# B&R Automation Studio project mappFramework (part 3)

### McBaseCfg.typ
```iecst
TYPE
	McCfgString250Type : STRING[250]; (**)
	McCfgTypeEnum :
		( (*Configuration system enum*)
		mcCFG_NONE := 0, (*None -*)
		mcCFG_MMCFG := 10, (*Associated with data type McCfgMMCfgType*)
		mcCFG_WS := 800, (*Associated with data type McCfgWorkspaceType*)
		mcCFG_TOOLTBL := 900, (*Tooltable -*)
		mcCFG_FRMTBL := 1000, (*Associated with data type McCfgFrmTblType*)
		mcCFG_DYNPARTBL := 1100, (**)
		mcCFG_TOOL := 1300, (*Tool -*)
		mcCFG_LIMSET_LIN := 1411, (*Associated with data type McCfgLimSetLinType*)
		mcCFG_LIMSET_ROT := 1412, (*Associated with data type McCfgLimSetRotType*)
		mcCFG_PROC_PT_LST := 1600, (*Associated with data type McCfgProcPtLstType*)
		mcCFG_AX := 10000, (*Associated with data type McCfgAxType*)
		mcCFG_AX_BASE_TYP := 10011, (*Associated with data type McCfgAxBaseTypType*)
		mcCFG_AX_MOVE_LIM := 10012, (*Associated with data type McCfgAxMoveLimType*)
		mcCFG_AX_FEAT_CAM_AUT_CMN := 10101, (*AxisFeatureCamAutCommon -*)
		mcCFG_AX_FEAT_PROF_GEN := 10102, (*AxisFeatureProfGen -*)
		mcCFG_AX_FEAT_DIG_CAM_SW := 10103, (*Associated with data type McCfgAxFeatDigCamSwType*)
		mcCFG_AX_FEAT_CAM_LST := 11102, (*AxisFeatureCamList -*)
		mcCFG_AX_FEAT_ALT_VAL_SRC := 10104, (*Associated with data type McCfgAxFeatAltValSrcType*)
		mcCFG_AX_FEAT_BRK := 10105, (*Associated with data type McCfgAxFeatBrkType*)
		mcCFG_AX_FEAT_MECH_DEV_COMP := 10106, (*Associated with data type McCfgAxFeatMechDevCompType*)
		mcCFG_MOT_SYN := 10500, (*Associated with data type McCfgMotSynType*)
		mcCFG_MOT_INDUCT := 10501, (*Associated with data type McCfgMotInductType*)
		mcCFG_IO_PL_IN_CARD := 10510, (*IOPlugInCard -*)
		mcCFG_ACP_AX := 11000, (*Associated with data type McCfgAcpAxType*)
		mcCFG_ACP_AX_REF := 11011, (*Associated with data type McCfgAcpAxRefType*)
		mcCFG_ACP_MECH_ELM := 11012, (*Associated with data type McCfgAcpMechElmType*)
		mcCFG_ACP_ENC_LINK := 11013, (*Associated with data type McCfgAcpEncLinkType*)
		mcCFG_ACP_CTRL := 11014, (*Associated with data type McCfgAcpCtrlType*)
		mcCFG_ACP_HOME := 11015, (*Associated with data type McCfgAcpHomeType*)
		mcCFG_ACP_STOP_REAC := 11016, (*Associated with data type McCfgAcpStopReacType*)
		mcCFG_ACP_MOVE_ERR_LIM := 11017, (*Associated with data type McCfgAcpMoveErrLimType*)
		mcCFG_ACP_JERK_FLTR := 11018, (*Associated with data type McCfgAcpJerkFltrType*)
		mcCFG_ACP_DIG_IN := 11019, (*Associated with data type McCfgAcpDigInType*)
		mcCFG_ACP_SIM := 11020, (*Associated with data type McCfgAcpSimType*)
		mcCFG_ACP_AX_FEAT := 11021, (*Associated with data type McCfgAcpAxFeatType*)
		mcCFG_ACP_AUX_PWR_SUP_MOD := 11030, (*Associated with data type McCfgAcpAuxPwrSupModType*)
		mcCFG_ACP_PSM_PWR_SEC := 11031, (*Associated with data type McCfgAcpPSMPwrSecType*)
		mcCFG_ACP_PWR_SUP := 11040, (*Associated with data type McCfgAcpPwrSupType*)
		mcCFG_ACP_ENC := 11045, (*Associated with data type McCfgAcpEncType*)
		mcCFG_ACP_VIRT_AX := 11050, (*Associated with data type McCfgAcpVirtAxType*)
		mcCFG_ACP_VIRT_AX_REF := 11051, (*Associated with data type McCfgAcpVirtAxRefType*)
		mcCFG_ACP_VIRT_HOME := 11052, (*Associated with data type McCfgAcpVirtHomeType*)
		mcCFG_ACP_VIRT_JERK_FLTR := 11053, (*Associated with data type McCfgAcpVirtJerkFltrType*)
		mcCFG_ACP_VIRT_AX_FEAT := 11054, (*Associated with data type McCfgAcpVirtAxFeatType*)
		mcCFG_ACP_CH_FEAT := 11060, (*Associated with data type McCfgAcpChFeatType*)
		mcCFG_ACP_EXT_ENC_AX := 11070, (*Associated with data type McCfgAcpExtEncAxType*)
		mcCFG_ACP_EXT_ENC_AX_REF := 11071, (*Associated with data type McCfgAcpExtEncAxRefType*)
		mcCFG_ACP_EXT_ENC_AX_ENC_LINK := 11072, (*Associated with data type McCfgAcpExtEncAxEncLinkType*)
		mcCFG_ACP_EXT_ENC_AX_MECH_ELM := 11073, (*Associated with data type McCfgAcpExtEncAxMechElmType*)
		mcCFG_ACP_EXT_ENC_AX_HOME := 11074, (*Associated with data type McCfgAcpExtEncAxHomeType*)
		mcCFG_AX_FEAT_CAM_AUT_ACP := 11101, (*AxisFeatureCamAutAcopos -*)
		mcCFG_AX_FEAT_A_IN := 11103, (*AxisFeatureAInput -*)
		mcCFG_AX_FEAT_ACP_PAR_TBL := 11104, (*Associated with data type McCfgAxFeatAcpParTblType*)
		mcCFG_PURE_V_AX := 12000, (*Associated with data type McCfgPureVAxType*)
		mcCFG_PURE_V_AX_REF := 12011, (*Associated with data type McCfgPureVAxRefType*)
		mcCFG_PURE_V_AX_HOME := 12012, (*Associated with data type McCfgPureVAxHomeType*)
		mcCFG_PURE_V_AX_JERK_FLTR := 12013, (*Associated with data type McCfgPureVAxJerkFltrType*)
		mcCFG_PURE_V_AX_FEAT := 12014, (*Associated with data type McCfgPureVAxFeatType*)
		mcCFG_PURE_V_AX_MECH_ELM := 12015, (*Associated with data type McCfgPureVAxMechElmType*)
		mcCFG_PURE_V_AX_ENC_LINK := 12016, (*Associated with data type McCfgPureVAxEncLinkType*)
		mcCFG_PURE_V_AX_CTRL := 12017, (*Associated with data type McCfgPureVAxCtrlType*)
		mcCFG_PURE_V_AX_STOP_REAC := 12018, (*Associated with data type McCfgPureVAxStopReacType*)
		mcCFG_PURE_V_AX_MOVE_ERR_LIM := 12019, (*Associated with data type McCfgPureVAxMoveErrLimType*)
		mcCFG_PURE_V_AX_DIG_IN := 12020, (*Associated with data type McCfgPureVAxDigInType*)
		mcCFG_PURE_V_AX_STAT_IN := 12021, (*Associated with data type McCfgPureVAxStatInType*)
		mcCFG_PURE_V_AX_CTRL_OUT := 12022, (*Associated with data type McCfgPureVAxCtrlOutType*)
		mcCFG_STP_AX := 13000, (*Associated with data type McCfgStpAxType*)
		mcCFG_STP_AX_REF := 13011, (*Associated with data type McCfgStpAxRefType*)
		mcCFG_STP_AX_MECH_ELM := 13012, (*Associated with data type McCfgStpAxMechElmType*)
		mcCFG_STP_AX_MOT := 13013, (*Associated with data type McCfgStpAxMotType*)
		mcCFG_STP_AX_ENC_LINK := 13014, (*Associated with data type McCfgStpAxEncLinkType*)
		mcCFG_STP_AX_CTRL := 13015, (*Associated with data type McCfgStpAxCtrlType*)
		mcCFG_STP_AX_HOME := 13016, (*Associated with data type McCfgStpAxHomeType*)
		mcCFG_STP_AX_STOP_REAC := 13017, (*Associated with data type McCfgStpAxStopReacType*)
		mcCFG_STP_AX_MOVE_ERR_LIM := 13018, (*Associated with data type McCfgStpAxMoveErrLimType*)
		mcCFG_STP_AX_JERK_FLTR := 13019, (*Associated with data type McCfgStpAxJerkFltrType*)
		mcCFG_STP_AX_DIG_IN := 13020, (*Associated with data type McCfgStpAxDigInType*)
		mcCFG_STP_AX_DIG_OUT := 13021, (*Associated with data type McCfgStpAxDigOutType*)
		mcCFG_STP_AX_FEAT := 13022, (*Associated with data type McCfgStpAxFeatType*)
		mcCFG_STP_ENC := 13100, (*Associated with data type McCfgStpEncType*)
		mcCFG_DS402_AX := 13500, (*Associated with data type McCfgDS402AxType*)
		mcCFG_DS402_INV_AX := 13501, (*Associated with data type McCfgDS402InvAxType*)
		mcCFG_DS402_AX_REF := 13511, (*Associated with data type McCfgDS402AxRefType*)
		mcCFG_DS402_AX_MECH_ELM := 13512, (*Associated with data type McCfgDS402AxMechElmType*)
		mcCFG_DS402_AX_ENC_SET := 13513, (*Associated with data type McCfgDS402AxEncSetType*)
		mcCFG_DS402_AX_POS_ACT_VAL_RNG := 13514, (*Associated with data type McCfgDS402AxPosActValRngType*)
		mcCFG_DS402_AX_CYC_SET_VAL_MOD := 13515, (*Associated with data type McCfgDS402AxCycSetValModType*)
		mcCFG_DS402_AX_FEAT := 13516, (*Associated with data type McCfgDS402AxFeatType*)
		mcCFG_ACP_INV_AX := 13600, (*Associated with data type McCfgAcpInvAxType*)
		mcCFG_ACP_INV_AX_REF := 13611, (*Associated with data type McCfgAcpInvAxRefType*)
		mcCFG_ACP_INV_AX_MECH_ELM := 13612, (*Associated with data type McCfgAcpInvAxMechElmType*)
		mcCFG_AXGRP_ADMIN := 20000, (*Associated with data type McCfgAxGrpAdminType*)
		mcCFG_AXGRP_FEAT_HOME_ORD := 20101, (*Associated with data type McCfgAxGrpFeatHomeOrdType*)
		mcCFG_AXGRP_FEAT_PWR_ON_ORD := 20102, (*Associated with data type McCfgAxGrpFeatPwrOnOrdType*)
		mcCFG_AXGRP_FEAT_EX_SNG_AX := 20103, (*Associated with data type McCfgAxGrpFeatExSngAxType*)
		mcCFG_AXGRP_FEAT_SHR_BRK_SIG := 20104, (*Associated with data type McCfgAxGrpFeatShrBrkSigType*)
		mcCFG_AXGRP_PATHGEN := 21000, (*Associated with data type McCfgAxGrpPathGenType*)
		mcCFG_AXGRP_PATHGEN_BASE_SET := 21013, (*Associated with data type McCfgAxGrpPathGenBaseSetType*)
		mcCFG_AXGRP_FEAT_PRG := 21101, (*Associated with data type McCfgAxGrpFeatPrgType*)
		mcCFG_AXGRP_FEAT_COMP := 21102, (*Associated with data type McCfgAxGrpFeatCompType*)
		mcCFG_AXGRP_FEAT_CDC := 21103, (*Associated with data type McCfgAxGrpFeatCdcType*)
		mcCFG_AXGRP_FEAT_FF := 21104, (*Associated with data type McCfgAxGrpFeatFfType*)
		mcCFG_AXGRP_FEAT_FRM_HIER_STD := 21105, (*Associated with data type McCfgAxGrpFeatFrmHierStdType*)
		mcCFG_AXGRP_FEAT_FRM_HIER_CUS := 21106, (*Associated with data type McCfgAxGrpFeatFrmHierCusType*)
		mcCFG_AXGRP_FEAT_JOG := 21107, (*AxesgroupFeatureJogging -*)
		mcCFG_AXGRP_FEAT_LAH := 21108, (*Associated with data type McCfgAxGrpFeatLahType*)
		mcCFG_AXGRP_FEAT_MFUN := 21109, (*Associated with data type McCfgAxGrpFeatMFunType*)
		mcCFG_AXGRP_FEAT_MON_ELEM := 21110, (*Associated with data type McCfgAxGrpFeatMonElemType*)
		mcCFG_AXGRP_FEAT_MP_LOG := 21111, (*Associated with data type McCfgAxGrpFeatMpLogType*)
		mcCFG_AXGRP_FEAT_PATH_DEF := 21112, (*Associated with data type McCfgAxGrpFeatPathDefType*)
		mcCFG_AXGRP_FEAT_PRG_SIM := 21113, (*Associated with data type McCfgAxGrpFeatPrgSimType*)
		mcCFG_AXGRP_FEAT_SPINDLES := 21114, (*Associated with data type McCfgAxGrpFeatSpindlesType*)
		mcCFG_AXGRP_FEAT_TOOL := 21115, (*Associated with data type McCfgAxGrpFeatToolType*)
		mcCFG_AXGRP_FEAT_WSM := 21116, (*Associated with data type McCfgAxGrpFeatWsmType*)
		mcCFG_AXGRP_FEAT_EX_PATH_AX := 21117, (*Associated with data type McCfgAxGrpFeatExPathAxType*)
		mcCFG_AXGRP_FEAT_PROBE := 21118, (*Associated with data type McCfgAxGrpFeatProbeType*)
		mcCFG_AXGRP_FEAT_SIG := 21119, (*Associated with data type McCfgAxGrpFeatSigType*)
		mcCFG_AXGRP_FEAT_2D_COMP := 21120, (*Associated with data type McCfgAxGrpFeat2DCompType*)
		mcCFG_AXGRP_FEAT_3D_COMP := 21121, (*Associated with data type McCfgAxGrpFeat3DCompType*)
		mcCFG_AXGRP_FEAT_PATH_PREVIEW := 21122, (*Associated with data type McCfgAxGrpFeatPathPreviewType*)
		mcCFG_AXGRP_FEAT_TAN_TOOL := 21124, (*Associated with data type McCfgAxGrpFeatTanToolType*)
		mcCFG_AXGRP_FEAT_REV_MOVE := 21125, (*Associated with data type McCfgAxGrpFeatRevMoveType*)
		mcCFG_ASM := 31000, (*Associated with data type McCfgAsmType*)
		mcCFG_ASM_FEAT_CPLG := 31101, (*Associated with data type McCfgAsmFeatCplgType*)
		mcCFG_ASM_FEAT_SIM_SH_DEF := 31102, (*Associated with data type McCfgAsmFeatSimShDefType*)
		mcCFG_ASM_FEAT_SH_TRACE := 31103, (*Associated with data type McCfgAsmFeatShTraceType*)
		mcCFG_ASM_FEAT_SH_AUT_ATT := 31104, (*Associated with data type McCfgAsmFeatShAutAttType*)
		mcCFG_ASM_FEAT_LOC_LIM := 31105, (*Associated with data type McCfgAsmFeatLocLimType*)
		mcCFG_ASM_FEAT_EX_SEG := 31106, (*Associated with data type McCfgAsmFeatExSegType*)
		mcCFG_ASM_FEAT_SH_SHP_REG := 31107, (*Associated with data type McCfgAsmFeatShShpRegType*)
		mcCFG_SEC_COMP := 31301, (*Associated with data type McCfgSecCompType*)
		mcCFG_SEC_SUB := 31302, (*Associated with data type McCfgSecSubType*)
		mcCFG_SH_STEREO_TYP := 31400, (*Associated with data type McCfgShStereoTypType*)
		mcCFG_SEG := 31500, (*Associated with data type McCfgSegType*)
		mcCFG_MS_CUS_STD := 50001, (*Associated with data type McCfgMSCusStdType*)
		mcCFG_MS_2AX_CNC_XY := 51201, (*Associated with data type McCfgMS2AxCncXYType*)
		mcCFG_MS_2AX_CNC_XZ := 51202, (*Associated with data type McCfgMS2AxCncXZType*)
		mcCFG_MS_2AX_CNC_YZ := 51203, (*Associated with data type McCfgMS2AxCncYZType*)
		mcCFG_MS_3AX_CNC_XYZ := 51301, (*Associated with data type McCfgMS3AxCncXYZType*)
		mcCFG_MS_3AX_CNC_XZC := 51302, (*Associated with data type McCfgMS3AxCncXZCType*)
		mcCFG_MS_3AX_CNC_XZB := 51303, (*Associated with data type McCfgMS3AxCncXZBType*)
		mcCFG_MS_4AX_CNC_XYZB := 51401, (*Associated with data type McCfgMS4AxCncXYZBType*)
		mcCFG_MS_4AX_CNC_XYZC := 51402, (*Associated with data type McCfgMS4AxCncXYZCType*)
		mcCFG_MS_5AX_CNC_XYZCA := 51504, (*Associated with data type McCfgMS5AxCncXYZCAType*)
		mcCFG_MS_6AX_CNC_ZXYBCA := 51603, (*Associated with data type McCfgMS6AxCncZXYBCAType*)
		mcCFG_MS_4AX_SCARA_A := 52041, (*Associated with data type McCfgMS4AxScaraAType*)
		mcCFG_MS_2AX_DELTA_A := 52121, (*Associated with data type McCfgMS2AxDeltaAType*)
		mcCFG_MS_3AX_DELTA_A := 52131, (*Associated with data type McCfgMS3AxDeltaAType*)
		mcCFG_MS_3AX_DELTA_XZB := 52132, (*Associated with data type McCfgMS3AxDeltaXZBType*)
		mcCFG_MS_3AX_DELTA_B := 52133, (*Associated with data type McCfgMS3AxDeltaBType*)
		mcCFG_MS_4AX_DELTA_A := 52141, (*Associated with data type McCfgMS4AxDeltaAType*)
		mcCFG_MS_4AX_DELTA_B := 52142, (*Associated with data type McCfgMS4AxDeltaBType*)
		mcCFG_MS_4AX_DELTA_C := 52143, (*Associated with data type McCfgMS4AxDeltaCType*)
		mcCFG_MS_5AX_DELTA_A := 52151, (*Associated with data type McCfgMS5AxDeltaAType*)
		mcCFG_MS_3AX_ROB_A := 52301, (*Associated with data type McCfgMS3AxRobAType*)
		mcCFG_MS_4AX_ROB_A := 52401, (*Associated with data type McCfgMS4AxRobAType*)
		mcCFG_MS_4AX_ROB_B := 52402, (*Associated with data type McCfgMS4AxRobBType*)
		mcCFG_MS_5AX_ROB_A := 52501, (*Associated with data type McCfgMS5AxRobAType*)
		mcCFG_MS_5AX_ROB_B := 52502, (*Associated with data type McCfgMS5AxRobBType*)
		mcCFG_MS_6AX_ROB_A := 52601, (*Associated with data type McCfgMS6AxRobAType*)
		mcCFG_MS_6AX_ROB_B := 52602, (*Associated with data type McCfgMS6AxRobBType*)
		mcCFG_MS_6AX_ROB_C := 52603 (*Associated with data type McCfgMS6AxRobCType*)
		);
	McCfgUnboundedArrayType : STRUCT (*General purpose datatype*)
		NumberOfElements : UDINT;
		DataAddress : UDINT;
		NumberOfArrayElements : UDINT;
	END_STRUCT;
	McCfgReferenceType : STRUCT (*General purpose datatype*)
		Name : STRING[250];
		ConfigType : McCfgTypeEnum;
	END_STRUCT;
	McMMCProcProcTskCEnum :
		( (*Cyclic task class for command processing*)
		mcMMCPPTC_CYC_1 := 1, (*Cyclic #1 - Task class 1*)
		mcMMCPPTC_CYC_2 := 2 (*Cyclic #2 - Task class 2*)
		);
	McMMCProcType : STRUCT
		ProcessingTaskClass : McMMCProcProcTskCEnum; (*Cyclic task class for command processing*)
	END_STRUCT;
	McMMCLogSelEnum :
		( (*Selective logging selector setting*)
		mcMMCLS_NOT_USE := 0, (*Not used -*)
		mcMMCLS_USE := 1 (*Used -*)
		);
	McCfgVisEnum :
		( (*Component state change logger entries (PLCopen state)*)
		mcCV_VIS := 0, (*Visible*)
		mcCV_SUP := 1 (*Suppressed*)
		);
	McMMCLogSelUseAdmCmdEnum :
		( (*Administrative commands selector setting*)
		mcMMCLSUAC_VIS := 0, (*Visible - This command group of logger entries will be visible*)
		mcMMCLSUAC_SUP := 1, (*Suppressed - This command group of logger entries will be suppressed*)
		mcMMCLSUAC_SEL := 2 (*Selective - Defines which sections of this command group should be visible*)
		);
	McMMCLogSelUseAdmCmdSelType : STRUCT (*Type mcMMCLSUAC_SEL settings*)
		CallerInstance : McCfgVisEnum; (*Logging of the caller instance entries*)
		ComponentResponse : McCfgVisEnum; (*Logging of component response entries*)
		AdditionalInformation : McCfgVisEnum; (*Logging of additional information entries*)
	END_STRUCT;
	McMMCLogSelUseAdmCmdType : STRUCT (*Administrative logger entries*)
		Type : McMMCLogSelUseAdmCmdEnum; (*Administrative commands selector setting*)
		Selective : McMMCLogSelUseAdmCmdSelType; (*Type mcMMCLSUAC_SEL settings*)
	END_STRUCT;
	McMMCLogSelUseMoveCmdEnum :
		( (*Movement commands selector setting*)
		mcMMCLSUMC_VIS := 0, (*Visible - This command group of logger entries will be visible*)
		mcMMCLSUMC_SUP := 1, (*Suppressed - This command group of logger entries will be suppressed*)
		mcMMCLSUMC_SEL := 2 (*Selective - Defines which sections of this command group should be visible*)
		);
	McMMCLogSelUseMoveCmdSelType : STRUCT (*Type mcMMCLSUMC_SEL settings*)
		CallerInstance : McCfgVisEnum; (*Logging of the caller instance entries*)
		ComponentResponse : McCfgVisEnum; (*Logging of component response entries*)
		AdditionalInformation : McCfgVisEnum; (*Logging of additional information entries*)
	END_STRUCT;
	McMMCLogSelUseMoveCmdType : STRUCT (*Movement logger entries*)
		Type : McMMCLogSelUseMoveCmdEnum; (*Movement commands selector setting*)
		Selective : McMMCLogSelUseMoveCmdSelType; (*Type mcMMCLSUMC_SEL settings*)
	END_STRUCT;
	McMMCLogSelUseInfoCmdEnum :
		( (*Informational commands selector setting*)
		mcMMCLSUIC_VIS := 0, (*Visible - This command group of logger entries will be visible*)
		mcMMCLSUIC_SUP := 1, (*Suppressed - This command group of logger entries will be suppressed*)
		mcMMCLSUIC_SEL := 2 (*Selective - Defines which sections of this command group should be visible*)
		);
	McMMCLogSelUseInfoCmdSelType : STRUCT (*Type mcMMCLSUIC_SEL settings*)
		CallerInstance : McCfgVisEnum; (*Logging of the caller instance entries*)
		ComponentResponse : McCfgVisEnum; (*Logging of component response entries*)
		AdditionalInformation : McCfgVisEnum; (*Logging of additional information entries*)
	END_STRUCT;
	McMMCLogSelUseInfoCmdType : STRUCT (*Status information logger entries*)
		Type : McMMCLogSelUseInfoCmdEnum; (*Informational commands selector setting*)
		Selective : McMMCLogSelUseInfoCmdSelType; (*Type mcMMCLSUIC_SEL settings*)
	END_STRUCT;
	McMMCLogSelUseSupSubcEEnum :
		( (*Suppress entries for internally invoked commands for subcomponents*)
		mcMMCLSUSSE_INACT := 0, (*Inactive - Entries for internally invoked commands for subcomponents are shown unless the base entries are suppressed*)
		mcMMCLSUSSE_ACT := 1 (*Active - Entries for internally invoked commands for subcomponents are suppressed*)
		);
	McMMCLogSelUseType : STRUCT (*Type mcMMCLS_USE settings*)
		StateChange : McCfgVisEnum; (*Component state change logger entries (PLCopen state)*)
		AdministrativeCommands : McMMCLogSelUseAdmCmdType; (*Administrative logger entries*)
		MovementCommands : McMMCLogSelUseMoveCmdType; (*Movement logger entries*)
		InformationalCommands : McMMCLogSelUseInfoCmdType; (*Status information logger entries*)
		SuppressSubcomponentEntries : McMMCLogSelUseSupSubcEEnum; (*Suppress entries for internally invoked commands for subcomponents*)
	END_STRUCT;
	McMMCLogSelType : STRUCT (*Define which logging areas should be visible*)
		Type : McMMCLogSelEnum; (*Selective logging selector setting*)
		Used : McMMCLogSelUseType; (*Type mcMMCLS_USE settings*)
	END_STRUCT;
	McMMCLogType : STRUCT
		Selective : McMMCLogSelType; (*Define which logging areas should be visible*)
	END_STRUCT;
	McCfgMMCfgType : STRUCT (*Main data type corresponding to McCfgTypeEnum mcCFG_MMCFG*)
		Processing : McMMCProcType;
		Logger : McMMCLogType;
	END_STRUCT;
	McCfgTransXYZType : STRUCT (*Translation parameters*)
		X : LREAL; (*Translation in X direction [measurement units]*)
		Y : LREAL; (*Translation in Y direction [measurement units]*)
		Z : LREAL; (*Translation in Z direction [measurement units]*)
	END_STRUCT;
	McCfgOrientType : STRUCT (*Orientation parameters*)
		Angle1 : LREAL; (*Rotation around the first coordinateaxis of the rotation order [measurement units]*)
		Angle2 : LREAL; (*Rotation around the second coordinateaxis of the rotation order [measurement units]*)
		Angle3 : LREAL; (*Rotation around the third coordinateaxis of the rotation order [measurement units]*)
	END_STRUCT;
	McWSCubeDimType : STRUCT (*Dimension parameters*)
		X : LREAL; (*Dimension of the cuboid in the x-direction (endpoint) [measurement units]*)
		Y : LREAL; (*Dimension of the cuboid in the y-direction (endpoint) [measurement units]*)
		Z : LREAL; (*Dimension of the cuboid in the z-direction (endpoint) [measurement units]*)
	END_STRUCT;
	McWSCubeType : STRUCT
		ID : UDINT; (*Unique cuboid ID*)
		Translation : McCfgTransXYZType; (*Translation parameters*)
		Orientation : McCfgOrientType; (*Orientation parameters*)
		Dimension : McWSCubeDimType; (*Dimension parameters*)
	END_STRUCT;
	McWSCubesType : STRUCT (*Defines cuboids*)
		Cuboid : McCfgUnboundedArrayType;
	END_STRUCT;
	McWSHalfSpcPlEnum :
		( (*Defines plane*)
		mcWSHSP_PL_XY := 0, (*Plane XY*)
		mcWSHSP_PL_YZ := 1, (*Plane YZ*)
		mcWSHSP_PL_ZX := 2 (*Plane ZX*)
		);
	McWSHalfSpcType : STRUCT
		ID : UDINT; (*Unique half-space ID*)
		Translation : McCfgTransXYZType; (*Translation parameters*)
		Orientation : McCfgOrientType; (*Orientation parameters*)
		Plane : McWSHalfSpcPlEnum; (*Defines plane*)
	END_STRUCT;
	McWSHalfSpcsType : STRUCT (*Defines half-spaces*)
		HalfSpace : McCfgUnboundedArrayType;
	END_STRUCT;
	McWSTcConeParType : STRUCT (*Object description parameters*)
		BaseRadius : LREAL; (*Base radius of the cone [measurement units]*)
		Height : LREAL; (*Height of the cone [measurement units]*)
		TopRadius : LREAL; (*Top radius of the cone [measurement units]*)
	END_STRUCT;
	McWSTcConeType : STRUCT (*Selects object type*)
		ID : UDINT; (*Unique object ID*)
		Translation : McCfgTransXYZType; (*Translation parameters*)
		Orientation : McCfgOrientType; (*Orientation parameters*)
		Parameters : McWSTcConeParType; (*Object description parameters*)
	END_STRUCT;
	McWSTcConesType : STRUCT (*Defines truncated cones*)
		TruncatedCone : McCfgUnboundedArrayType; (*Selects object type*)
	END_STRUCT;
	McWSWorkSpaceType : STRUCT (*Defines the WorkSpace*)
		Cuboids : McWSCubesType; (*Defines cuboids*)
		HalfSpaces : McWSHalfSpcsType; (*Defines half-spaces*)
		TruncatedCones : McWSTcConesType; (*Defines truncated cones*)
	END_STRUCT;
	McWSSafeSpaceType : STRUCT (*Defines the SafeSpace*)
		Cuboids : McWSCubesType; (*Defines cuboids*)
		HalfSpaces : McWSHalfSpcsType; (*Defines half-spaces*)
		TruncatedCones : McWSTcConesType; (*Defines truncated cones*)
	END_STRUCT;
	McCfgWorkspaceType : STRUCT (*Main data type corresponding to McCfgTypeEnum mcCFG_WS*)
		WorkSpace : McWSWorkSpaceType; (*Defines the WorkSpace*)
		SafeSpace : McWSSafeSpaceType; (*Defines the SafeSpace*)
	END_STRUCT;
	McFTRowType : STRUCT
		Index : UINT;
		X : LREAL;
		Y : LREAL;
		Z : LREAL;
		Angle1 : LREAL;
		Angle2 : LREAL;
		Angle3 : LREAL;
		Description : STRING[250];
	END_STRUCT;
	McCfgFrmTblType : STRUCT (*Main data type corresponding to McCfgTypeEnum mcCFG_FRMTBL*)
		Row : McCfgUnboundedArrayType;
	END_STRUCT;
	McLSPosEnum :
		( (*Position selector setting*)
		mcLSP_NOT_USE := 0, (*Not used -*)
		mcLSP_USE := 1 (*Used -*)
		);
	McCfgLimPosType : STRUCT (*Type mcLSP_USE settings*)
		LowerLimit : LREAL; (*Lower software limit position [Measurement units]*)
		UpperLimit : LREAL; (*Upper software limit position [Measurement units]*)
	END_STRUCT;
	McLSPosType : STRUCT (*Movement range of the axis via two position boundaries*)
		Type : McLSPosEnum; (*Position selector setting*)
		Used : McCfgLimPosType; (*Type mcLSP_USE settings*)
	END_STRUCT;
	McLSVelEnum :
		( (*Velocity selector setting*)
		mcLSV_NOT_USE := 0, (*Not used -*)
		mcLSV_BASIC := 1, (*Basic -*)
		mcLSV_ADV := 2 (*Advanced -*)
		);
	McCfgLimVelBaseType : STRUCT (*Type mcLSV_BASIC settings*)
		Velocity : REAL; (*Velocity limit in any movement direction [Measurement units/s]*)
	END_STRUCT;
	McCfgLimVelAdvType : STRUCT (*Type mcLSV_ADV settings*)
		Positive : REAL; (*Velocity limit in positive movement direction [Measurement units/s]*)
		Negative : REAL; (*Velocity limit in negative movement direction [Measurement units/s]*)
	END_STRUCT;
	McLSVelType : STRUCT (*Velocity limits*)
		Type : McLSVelEnum; (*Velocity selector setting*)
		Basic : McCfgLimVelBaseType; (*Type mcLSV_BASIC settings*)
		Advanced : McCfgLimVelAdvType; (*Type mcLSV_ADV settings*)
	END_STRUCT;
	McLSAccEnum :
		( (*Acceleration selector setting*)
		mcLSA_NOT_USE := 0, (*Not used -*)
		mcLSA_BASIC := 1, (*Basic -*)
		mcLSA_ADV := 2 (*Advanced -*)
		);
	McCfgLimAccBaseType : STRUCT (*Type mcLSA_BASIC settings*)
		Acceleration : REAL; (*Acceleration limit in any movement direction [Measurement units/s²]*)
	END_STRUCT;
	McCfgLimAccAdvType : STRUCT (*Type mcLSA_ADV settings*)
		Positive : REAL; (*Acceleration limit in positive movement direction [Measurement units/s²]*)
		Negative : REAL; (*Acceleration limit in negative movement direction [Measurement units/s²]*)
	END_STRUCT;
	McLSAccType : STRUCT (*Acceleration limits*)
		Type : McLSAccEnum; (*Acceleration selector setting*)
		Basic : McCfgLimAccBaseType; (*Type mcLSA_BASIC settings*)
		Advanced : McCfgLimAccAdvType; (*Type mcLSA_ADV settings*)
	END_STRUCT;
	McLSDecEnum :
		( (*Deceleration selector setting*)
		mcLSD_NOT_USE := 0, (*Not used -*)
		mcLSD_BASIC := 1, (*Basic -*)
		mcLSD_ADV := 2 (*Advanced -*)
		);
	McCfgLimDecBaseType : STRUCT (*Type mcLSD_BASIC settings*)
		Deceleration : REAL; (*Deceleration limit in any movement direction [Measurement units/s²]*)
	END_STRUCT;
	McCfgLimDecAdvType : STRUCT (*Type mcLSD_ADV settings*)
		Positive : REAL; (*Deceleration limit in positive movement direction [Measurement units/s²]*)
		Negative : REAL; (*Deceleration limit in negative movement direction [Measurement units/s²]*)
	END_STRUCT;
	McLSDecType : STRUCT (*Deceleration limits*)
		Type : McLSDecEnum; (*Deceleration selector setting*)
		Basic : McCfgLimDecBaseType; (*Type mcLSD_BASIC settings*)
		Advanced : McCfgLimDecAdvType; (*Type mcLSD_ADV settings*)
	END_STRUCT;
	McCfgLimJerkEnum :
		( (*Jerk selector setting*)
		mcCLJ_NOT_USE := 0, (*Not used -*)
		mcCLJ_BASIC := 1, (*Basic -*)
		mcCLJ_ADV := 2 (*Advanced -*)
		);
	McCfgLimJerkBasicType : STRUCT (*Type mcCLJ_BASIC settings*)
		Jerk : REAL; (*Jerk limit in any movement direction [Measurement units/s³]*)
	END_STRUCT;
	McCfgLimJerkAdvType : STRUCT (*Type mcCLJ_ADV settings*)
		AccelerationPositive : REAL; (*Jerk limit in positive movement direction during acceleration [Measurement units/s³]*)
		AccelerationNegative : REAL; (*Jerk limit in negative movement direction during acceleration [Measurement units/s³]*)
		DecelerationPositive : REAL; (*Jerk limit in positive movement direction during deceleration [Measurement units/s³]*)
		DecelerationNegative : REAL; (*Jerk limit in negative movement direction during deceleration [Measurement units/s³]*)
	END_STRUCT;
	McCfgLimJerkType : STRUCT (*Jerk limits*)
		Type : McCfgLimJerkEnum; (*Jerk selector setting*)
		Basic : McCfgLimJerkBasicType; (*Type mcCLJ_BASIC settings*)
		Advanced : McCfgLimJerkAdvType; (*Type mcCLJ_ADV settings*)
	END_STRUCT;
	McCfgLimForEnum :
		( (*Force selector setting*)
		mcCLF_NOT_USE := 0, (*Not used -*)
		mcCLF_BASIC := 1, (*Basic -*)
		mcCLF_ADV := 2 (*Advanced -*)
		);
	McCfgLimForBasicType : STRUCT (*Type mcCLF_BASIC settings*)
		Force : REAL; (*Force limit in any movement direction [N]*)
	END_STRUCT;
	McCfgLimForAdvType : STRUCT (*Type mcCLF_ADV settings*)
		AccelerationPositive : REAL; (*Force limit in positive movement direction during acceleration [N]*)
		AccelerationNegative : REAL; (*Force limit in negative movement direction during acceleration [N]*)
		DecelerationPositive : REAL; (*Force limit in positive movement direction during deceleration [N]*)
		DecelerationNegative : REAL; (*Force limit in negative movement direction during deceleration [N]*)
	END_STRUCT;
	McCfgLimForType : STRUCT (*Limits for the force of the axis*)
		Type : McCfgLimForEnum; (*Force selector setting*)
		Basic : McCfgLimForBasicType; (*Type mcCLF_BASIC settings*)
		Advanced : McCfgLimForAdvType; (*Type mcCLF_ADV settings*)
	END_STRUCT;
	McCfgLimSetLinType : STRUCT (*Main data type corresponding to McCfgTypeEnum mcCFG_LIMSET_LIN*)
		Position : McLSPosType; (*Movement range of the axis via two position boundaries*)
		Velocity : McLSVelType; (*Velocity limits*)
		Acceleration : McLSAccType; (*Acceleration limits*)
		Deceleration : McLSDecType; (*Deceleration limits*)
		Jerk : McCfgLimJerkType; (*Jerk limits*)
		Force : McCfgLimForType; (*Limits for the force of the axis*)
	END_STRUCT;
	McCfgLimTorqEnum :
		( (*Torque selector setting*)
		mcCLT_NOT_USE := 0, (*Not used -*)
		mcCLT_BASIC := 1, (*Basic -*)
		mcCLT_ADV := 2 (*Advanced -*)
		);
	McCfgLimTorqBasicType : STRUCT (*Type mcCLT_BASIC settings*)
		Torque : REAL; (*Torque limit in any movement direction [Nm]*)
	END_STRUCT;
	McCfgLimTorqAdvType : STRUCT (*Type mcCLT_ADV settings*)
		AccelerationPositive : REAL; (*Torque limit in positive movement direction during acceleration [Nm]*)
		AccelerationNegative : REAL; (*Torque limit in negative movement direction during acceleration [Nm]*)
		DecelerationPositive : REAL; (*Torque limit in positive movement direction during deceleration [Nm]*)
		DecelerationNegative : REAL; (*Torque limit in negative movement direction during deceleration [Nm]*)
	END_STRUCT;
	McCfgLimTorqType : STRUCT (*Torque limits*)
		Type : McCfgLimTorqEnum; (*Torque selector setting*)
		Basic : McCfgLimTorqBasicType; (*Type mcCLT_BASIC settings*)
		Advanced : McCfgLimTorqAdvType; (*Type mcCLT_ADV settings*)
	END_STRUCT;
	McCfgLimSetRotType : STRUCT (*Main data type corresponding to McCfgTypeEnum mcCFG_LIMSET_ROT*)
		Position : McLSPosType; (*Movement range of the axis via two position boundaries*)
		Velocity : McLSVelType; (*Velocity limits*)
		Acceleration : McLSAccType; (*Acceleration limits*)
		Deceleration : McLSDecType; (*Deceleration limits*)
		Jerk : McCfgLimJerkType; (*Jerk limits*)
		Torque : McCfgLimTorqType; (*Torque limits*)
	END_STRUCT;
	McPPLPtEnum :
		( (*Process point: {/} selector setting*)
		mcPPLP_TRAK_PT := 0 (*Trak point - ACOPOSTrak*)
		);
	McPPLPtTrakPtPosRelToEnum :
		( (*Absolute position from which the position is counted*)
		mcPPLPTPPRT_ST_OF_SEC := 0, (*Start of sector - Tail of the sector*)
		mcPPLPTPPRT_END_OF_SEC := 1 (*End of sector - Head of the sector*)
		);
	McPPLPtTrakPtBarrFunEnum :
		( (*Barrier functionality selector setting*)
		mcPPLPTPBF_OFF := 0, (*Off - Disable barrier functionality*)
		mcPPLPTPBF_ON := 1 (*On - Enable barrier functionality*)
		);
	McPPLPtTrakPtBarrFunType : STRUCT (*Enable barrier functionality for process point*)
		Type : McPPLPtTrakPtBarrFunEnum; (*Barrier functionality selector setting*)
	END_STRUCT;
	McPPLPtTrakPtType : STRUCT (*Type mcPPLP_TRAK_PT settings*)
		Name : STRING[250]; (*Identifier of point*)
		SectorReference : McCfgReferenceType; (*Name of the referenced sector component*)
		Position : LREAL; (*Position on the sector [Measurement units]*)
		PositionRelativeTo : McPPLPtTrakPtPosRelToEnum; (*Absolute position from which the position is counted*)
		TriggerEventBufferSize : UINT; (*Amount of maximum saved trigger point events*)
		BarrierFunctionality : McPPLPtTrakPtBarrFunType; (*Enable barrier functionality for process point*)
	END_STRUCT;
	McPPLPtType : STRUCT
		Type : McPPLPtEnum; (*Process point: {/} selector setting*)
		TrakPoint : McPPLPtTrakPtType; (*Type mcPPLP_TRAK_PT settings*)
	END_STRUCT;
	McCfgProcPtLstType : STRUCT (*Main data type corresponding to McCfgTypeEnum mcCFG_PROC_PT_LST*)
		ProcessPoints : McCfgUnboundedArrayType;
	END_STRUCT;
	McCfgLocLenUnitEnum :
		( (*Measurement unit for the axis*)
		mcCLLU_G_SET := 0, (*Global settings*)
		mcCLLU_MILL := 5066068, (*Millimeters*)
		mcCLLU_M := 5067858, (*Meters*)
		mcCLLU_INCH := 4804168, (*Inches*)
		mcCLLU_GEN := -1 (*Generic*)
		);
	McCfgCntDirEnum :
		( (*Direction of the axis in which the position value is increasing*)
		mcCCD_STD := 0, (*Standard - Rotary axis: clockwise*)
		mcCCD_INV := 1 (*Inverse - Rotary axis: counter-clockwise*)
		);
	McCfgLocRotUnitEnum :
		( (*Measurement unit for the axis*)
		mcCLRU_G_SET := 0, (*Global settings*)
		mcCLRU_DEG := 17476, (*Degrees*)
		mcCLRU_GRAD := 4274481, (*Gradians*)
		mcCLRU_REV := 5059636, (*Revolutions*)
		mcCLRU_GEN := -1 (*Generic*)
		);
	McCfgExtLimRefType : STRUCT (*Type mcAML_EXT settings*)
		LimitReference : McCfgReferenceType; (*Name of the limit reference*)
	END_STRUCT;
	McCfgGearBoxType : STRUCT (*Ratio between a gearbox input and output*)
		Input : DINT; (*Number of rotations on the encoder side [Revolutions]*)
		Output : DINT; (*Number of rotations on the load side which correspond to the number of rotations on the encoder side [Revolutions]*)
	END_STRUCT;
	McCfgRotToLinTrfType : STRUCT (*Specifies a transformation factor between the output of the gear and the actual load movement*)
		ReferenceDistance : LREAL; (*Reference distance which is considered for an axis positioning [Measurement units/Gearbox output revolution]*)
	END_STRUCT;
	McPTCEnum :
		( (*Cyclic task class for command processing*)
		mcPTC_CYC_1 := 1, (*Cyclic #1 - Task class 1*)
		mcPTC_USE_MP_MOT_SET := 255 (*Use mapp Motion setting - Use the defined setting from the mapp Motion configuration or Task class 1 if no mapp Motion Configuration exists*)
		);
	McCfgVarDatTypEnum :
		( (*Data type selector setting*)
		mcCVDT_TYP_BOOL := 0, (*Type BOOL -*)
		mcCVDT_TYP_SINT := 1, (*Type SINT -*)
		mcCVDT_TYP_USINT := 2, (*Type USINT -*)
		mcCVDT_TYP_INT := 3, (*Type INT -*)
		mcCVDT_TYP_UINT := 4, (*Type UINT -*)
		mcCVDT_TYP_DINT := 5, (*Type DINT -*)
		mcCVDT_TYP_UDINT := 6, (*Type UDINT -*)
		mcCVDT_TYP_REAL := 7, (*Type REAL -*)
		mcCVDT_TYP_LREAL := 8, (*Type LREAL -*)
		mcCVDT_TYP_STRING := 9, (*Type STRING -*)
		mcCVDT_TYP_DER := 10 (*Type Derived - Derived data type*)
		);
	McCfgVarDatTypTypSTRINGType : STRUCT (*Type mcCVDT_TYP_STRING settings*)
		Length : UDINT;
	END_STRUCT;
	McCfgVarDatTypTypDerType : STRUCT (*Type mcCVDT_TYP_DER settings*)
		Name : STRING[250]; (*Name*)
	END_STRUCT;
	McCfgVarDatTypType : STRUCT (*Data type*)
		Type : McCfgVarDatTypEnum; (*Data type selector setting*)
		TypeSTRING : McCfgVarDatTypTypSTRINGType; (*Type mcCVDT_TYP_STRING settings*)
		TypeDerived : McCfgVarDatTypTypDerType; (*Type mcCVDT_TYP_DER settings*)
	END_STRUCT;
	McCfgLimJerkBaseType : STRUCT (*Type mcAGFPDPLIJ_BASIC settings*)
		Jerk : REAL; (*Jerk limit in any movement direction [Measurement units/s³]*)
	END_STRUCT;
	McCfgTransXType : STRUCT (*Translation from base to QX*)
		X : LREAL; (*Translation in X direction [measurement units]*)
	END_STRUCT;
	McCfgTransZType : STRUCT (*Translation from QX to QZ*)
		Z : LREAL; (*Translation in Z direction [measurement units]*)
	END_STRUCT;
	McCfgTransXZType : STRUCT (*Translation from QZ to QB*)
		X : LREAL; (*Translation in X direction [measurement units]*)
		Z : LREAL; (*Translation in Z direction [measurement units]*)
	END_STRUCT;
	McCfgTransYType : STRUCT (*Translation from QX to QY*)
		Y : LREAL; (*Translation in Y direction [measurement units]*)
	END_STRUCT;
END_TYPE
```

### Program Logical/MachineControl/AppAxis_1/AppAxis_1

#### AxisMgr.typ
```iecst
(*Structure types*)

TYPE
	AxisSettingsType : 	STRUCT
		AxisFeatures : {REDUND_UNREPLICABLE} ARRAY[0..2]OF STRING[255]; (*Variable to write axis features into*)
		DriveConfiguration : {REDUND_UNREPLICABLE} McCfgPureVAxType; (*Drive configuration structure*)
		BaseConfiguration : {REDUND_UNREPLICABLE} McCfgAxType; (*Base axis type configuration *)
		BaseParam : {REDUND_UNREPLICABLE} McCfgAxMoveLimType; (*Base axis movement configuration*)
	END_STRUCT;
	AxisMachineSettingsType : {REDUND_UNREPLICABLE} 	STRUCT
		ReferencePosition : {REDUND_UNREPLICABLE} LREAL := 0; (*[mm] Axis position after reference*)
	END_STRUCT;
	AxisControlCommandType : {REDUND_UNREPLICABLE} 	STRUCT
		UpdatePreviewParameters : {REDUND_UNREPLICABLE} BOOL; (*Cmd to load new preview*)
		LoadRecipeParameters : {REDUND_UNREPLICABLE} BOOL; (*Load selected recipe file into active parameters *)
		SaveRecipeParameters : {REDUND_UNREPLICABLE} BOOL; (*Save current parameters*)
		Power : {REDUND_UNREPLICABLE} BOOL; (*Cmd power*)
		Reference : {REDUND_UNREPLICABLE} BOOL; (*Cmd home / reference*)
		MoveAbsolute : {REDUND_UNREPLICABLE} BOOL; (*Cmd move absolute*)
		MoveAdditive : {REDUND_UNREPLICABLE} BOOL; (*Cmd move additive*)
		MoveToStart : {REDUND_UNREPLICABLE} BOOL; (*Cmd move the start position*)
		Abort : {REDUND_UNREPLICABLE} BOOL; (*Cmd abort*)
		Stop : {REDUND_UNREPLICABLE} BOOL; (*Cmd stop all movement*)
		Reset : {REDUND_UNREPLICABLE} BOOL; (*Cmd reset axis state*)
		JogPositive : {REDUND_UNREPLICABLE} BOOL; (*Cmd jog positive*)
		JogNegative : {REDUND_UNREPLICABLE} BOOL; (*Cmd jog negative*)
		Start : {REDUND_UNREPLICABLE} BOOL; (*Cmd start motion*)
	END_STRUCT;
	AxisControlParametersType : {REDUND_UNREPLICABLE} 	STRUCT
		HomePosition : {REDUND_UNREPLICABLE} LREAL := 0; (*[mm] Home Position*)
		Position : {REDUND_UNREPLICABLE} LREAL := 0; (*[mm] Position for absolute move*)
		Distance : {REDUND_UNREPLICABLE} LREAL := 50; (*[mm] Distance for relative move*)
		Velocity : {REDUND_UNREPLICABLE} REAL := 100; (*[mm/s] Velocity for absoluate and relative moves*)
		Acceleration : {REDUND_UNREPLICABLE} REAL := 360; (*[mm/s2] Acceleration for absoluate and relative moves*)
		Deceleration : {REDUND_UNREPLICABLE} REAL := 360; (*[mm/s2] Deceleration for absoluate and relative moves*)
		JogVelocity : {REDUND_UNREPLICABLE} REAL := 100; (*[mm/s] Velocity used when jogging the axis*)
		StopDeceleration : {REDUND_UNREPLICABLE} REAL := 720; (*[mm/s2] Deceleration for stopping*)
		ProductNumber : {REDUND_UNREPLICABLE} INT := 0; (*Product Number*)
		ProductLength : {REDUND_UNREPLICABLE} REAL := 70; (*Real Product Length*)
	END_STRUCT;
	AxisControlStatusType : {REDUND_UNREPLICABLE} 	STRUCT
		TaskName : {REDUND_UNREPLICABLE} STRING[80]; (*Current task name for configuration changes*)
		MachineSettingsName : {REDUND_UNREPLICABLE} STRING[255]; (*Category name for machine settings*)
		ProductSettingsName : {REDUND_UNREPLICABLE} STRING[255]; (*Category name for product settings*)
		Status : {REDUND_UNREPLICABLE} STRING[80]; (*Machine Status*)
		IsReady : {REDUND_UNREPLICABLE} BOOL; (*Axis is ready*)
		ErrorActive : {REDUND_UNREPLICABLE} BOOL; (*Error active*)
		Busy : {REDUND_UNREPLICABLE} BOOL; (*Cmd execution*)
		ReferenceRequired : {REDUND_UNREPLICABLE} BOOL; (*Reference cmd required*)
		Position : {REDUND_UNREPLICABLE} LREAL; (*Current position*)
		Velocity : {REDUND_UNREPLICABLE} REAL; (*Current position*)
		Current : {REDUND_UNREPLICABLE} REAL; (*Drive current*)
		LagError : {REDUND_UNREPLICABLE} LREAL; (*Axis lag error *)
		MotorTemperature : {REDUND_UNREPLICABLE} REAL; (*Motor temperature*)
		IsHomed : {REDUND_UNREPLICABLE} BOOL; (*Axis is referenced*)
		IsPowered : {REDUND_UNREPLICABLE} BOOL; (*Axis is powered*)
	END_STRUCT;
	AxisControlType : {REDUND_UNREPLICABLE} 	STRUCT
		Command : {REDUND_UNREPLICABLE} AxisControlCommandType; (*Cmd structure*)
		Parameters : {REDUND_UNREPLICABLE} AxisControlParametersType; (*Parameter structure*)
		Status : {REDUND_UNREPLICABLE} AxisControlStatusType; (*Status structure*)
	END_STRUCT;
	AxisRecipeType : 	STRUCT
		EditDialogOpened : BOOL; (*HMI edit dialog open*)
		CreateDialogOpened : BOOL; (*HMI create dialog open*)
		SaveRecipe : BOOL; (*Cmd save current values*)
		LoadRecipe : BOOL; (*Cmd load exiting recipe*)
		CreateRecipe : BOOL; (*Cmd create new recipe*)
		State : AxisRecipeStepEnum; (*Recipe handling state*)
		CategoryDropdown : STRING[50]; (*HMI selector*)
	END_STRUCT;
END_TYPE

(*Enumerations*)

TYPE
	StateEnum :
		(
		STATE_INIT, (*Axis initialization state*)
		STATE_POWER_ON, (*Axis powering on state*)
		STATE_HOME, (*Axis homing state*)
		STATE_REFERENCE, (*Axis reference state*)
		STATE_MOVE_TO_HOME_POSITION, (*Axis moving to reference position state*)
		STATE_READY, (*Axis ready state*)
		STATE_MANUAL_OPERATION, (*Axis manual state*)
		STATE_AUTOMATIC_OPERATION, (*Axis automatic state*)
		STATE_STOPPING, (*Axis stopping state*)
		STATE_STOPPED, (*Axis stopped state*)
		STATE_ABORTING, (*Axis aborting state*)
		STATE_ABORTED, (*Axis aborted state*)
		STATE_CLEARING, (*Axis clearing state*)
		STATE_RESETTING (*Axis resetting state*)
		);
	ParameterStateEnum :
		(
		PAR_STATE_INIT, (*Param initialization state*)
		PAR_STATE_READ, (*Param read state*)
		PAR_STATE_WRITE, (*Param write state*)
		PAR_STATE_READY (*Param ready state*)
		);
	ConfigurationStateEnum :
		(
		CONFIG_STATE_INIT, (*Config initialization state*)
		CONFIG_STATE_READ, (*Config read state*)
		CONFIG_STATE_WRITE, (*Config write state*)
		CONFIG_STATE_READY (*Config ready state*)
		);
	ManualStateEnum :
		(
		MANUAL_STATE_IDLE, (*Idle state*)
		MANUAL_STATE_JOG, (*Jog state*)
		MANUAL_STATE_MOVE, (*Move state*)
		MANUAL_STATE_STOPPING (*Stopping state*)
		);
	AutomaticStateEnum :
		(
		AUTOMATIC_STATE_IDLE, (*Idle state*)
		AUTOMATIC_STATE_RUNNING (*Run state*)
		);
	AxisRecipeStepEnum :
		(
		REC_AXIS_WAIT, (*Wait state*)
		REC_AXIS_LOAD, (*Load product parameters*)
		REC_AXIS_SAVE, (*Save product parameters*)
		REC_AXIS_CREATE, (*Create new axis recipe*)
		REC_AXIS_STORE_MACH_SETTINGS, (*Save machine parameter settings*)
		REC_AXIS_FACTORY_RESET (*Factory reset*)
		);
END_TYPE
```

#### AxisControlModes.st
```iecst
ACTION AxisInit:
    // Action call during init
END_ACTION

ACTION AxisCyclic:
    // Cyclic action call
    MpAlarmXControl_SpeedNotSet.MpLink := ADR(gMpLinkAlarmXCoreAppAxis_1);
    MpAlarmXControl_SpeedNotSet.Enable := TRUE;
    MpAlarmXControl_SpeedNotSet.Name := ADR('AppAxis_1SpeedNotSet');
    MpAlarmXControl_SpeedNotSet();
    MpAlarmXControl_SpeedNotSet.Reset := FALSE;

END_ACTION

ACTION AxisManual:
    // Action handling manual axis control
    MpAxisParameters.Jog.Velocity := AxisControl.Parameters.JogVelocity;
    MpAxisParameters.Position := AxisControl.Parameters.Position;
    MpAxisParameters.Distance := AxisControl.Parameters.Distance;
    MpAxisParameters.Acceleration := AxisControl.Parameters.Acceleration;
    MpAxisParameters.Deceleration := AxisControl.Parameters.Deceleration;

    CASE ManualState OF
	// Wait state
        MANUAL_STATE_IDLE:
            IF ((AxisControl.Command.JogNegative = TRUE) OR (AxisControl.Command.JogPositive = TRUE)) THEN
                ManualState := MANUAL_STATE_JOG;
            ELSIF ((AxisControl.Command.MoveAbsolute = TRUE) OR (AxisControl.Command.MoveAdditive = TRUE)) THEN
                MpAxisBasic_0.MoveAbsolute := AxisControl.Command.MoveAbsolute;
                MpAxisBasic_0.MoveAdditive := AxisControl.Command.MoveAdditive;
                AxisControl.Command.MoveAbsolute := FALSE;
                AxisControl.Command.MoveAdditive := FALSE;
                ManualState := MANUAL_STATE_MOVE;
            END_IF
        // Jog state
        MANUAL_STATE_JOG:
            MpAxisBasic_0.JogNegative := AxisControl.Command.JogNegative;
            MpAxisBasic_0.JogPositive := AxisControl.Command.JogPositive;
            IF (AxisControl.Command.Stop = TRUE) THEN
                AxisControl.Command.Stop := FALSE;
                MpAxisBasic_0.Stop := TRUE;
                ManualState := MANUAL_STATE_STOPPING;
            ELSIF ((AxisControl.Command.JogNegative = FALSE) AND (AxisControl.Command.JogPositive = FALSE)) THEN
                MpAxisBasic_0.Stop := FALSE;
                MpAxisBasic_0.JogPositive := FALSE;
                MpAxisBasic_0.JogNegative := FALSE;
                ManualState := MANUAL_STATE_STOPPING;
            END_IF
       // Direct move state
        MANUAL_STATE_MOVE:
            IF (AxisControl.Command.Stop = TRUE) THEN
                MpAxisBasic_0.MoveAbsolute := FALSE;
                MpAxisBasic_0.MoveAdditive := FALSE;
                AxisControl.Command.Stop := FALSE;
                MpAxisBasic_0.Stop := TRUE;
                ManualState := MANUAL_STATE_STOPPING;
            ELSIF (InPositionEdgePos.Q = TRUE) THEN
                MpAxisBasic_0.MoveAbsolute := FALSE;
                MpAxisBasic_0.MoveAdditive := FALSE;
                ManualState := MANUAL_STATE_IDLE;
                State := STATE_READY;
            ELSIF ((AxisControl.Command.JogNegative = TRUE) OR (AxisControl.Command.JogPositive = TRUE)) THEN
                MpAxisBasic_0.MoveAbsolute := FALSE;
                MpAxisBasic_0.MoveAdditive := FALSE;
                ManualState := MANUAL_STATE_JOG;
            END_IF
        // Stopping active movements
        MANUAL_STATE_STOPPING:
            MpAxisBasic_0.JogNegative := FALSE;
            MpAxisBasic_0.JogPositive := FALSE;
            MpAxisBasic_0.MoveAbsolute := FALSE;
            MpAxisBasic_0.MoveAdditive := FALSE;

            IF (MpAxisBasic_0.MoveActive = FALSE) THEN
                ManualState := MANUAL_STATE_IDLE;
                State := STATE_READY;
            END_IF
    END_CASE

END_ACTION

ACTION AxisAutomatic:

    CASE AutomaticState OF
        AUTOMATIC_STATE_IDLE:
            IF (AxisControl.Command.Start = TRUE) THEN
                MpAlarmXControl_SpeedNotSet.Set := (MpAxisParameters.Velocity = 0);
                AxisControl.Command.Start := FALSE;
                AutomaticState := AUTOMATIC_STATE_RUNNING;
            END_IF

        AUTOMATIC_STATE_RUNNING:
            MpAxisBasic_0.MoveVelocity := TRUE;
            MpAxisParameters.Velocity := AxisControl.Parameters.Velocity;
            MpAxisParameters.Acceleration := AxisControl.Parameters.Acceleration;
            MpAxisParameters.Deceleration := AxisControl.Parameters.Deceleration;

            IF (AxisControl.Command.Stop = TRUE) THEN
                AxisControl.Command.Stop := FALSE;
                MpAxisBasic_0.MoveVelocity := FALSE;
                State := STATE_READY;
                AutomaticState := AUTOMATIC_STATE_IDLE;
            END_IF
    END_CASE

END_ACTION

ACTION AxisReset:

//    edge alarms don't require a reset
//    IF (MpAlarmXControl_SpeedNotSet.Set = TRUE) THEN
//        MpAlarmXControl_SpeedNotSet.Set := FALSE;
//        MpAlarmXControl_SpeedNotSet.ID := MpAlarmXControl_SpeedNotSet.InstanceID;
//        MpAlarmXControl_SpeedNotSet.Reset := TRUE;
//    END_IF

END_ACTION
```

### Program Logical/MachineControl/AppAxis_1/UnitTests/ConvTest (ANSIC)

#### TestType.typ
```iecst
TYPE
	testState_enum :
		(
		TEST_STATE_ARRANGE,
		TEST_STATE_ACT,
		TEST_STATE_ASSERT,
		TEST_STATE_DONE
		);
END_TYPE
```

#### autoGeneratedFile.c - Auto generated code - list of all test sets in the program
```c
/*
B+R UnitTest: This is generated code.
Do not edit! Do not move!
Description: UnitTest Testprogramm infrastructure (List of TestSets).
LastUpdated: 2021-09-27 19:12:47Z
By B+R UnitTest Helper Version: 2.0.1.59
*/
#include "UnitTest.h"

UNITTEST_TESTSET_DECLARATION  Set_SetupTeardown;

UNITTEST_TESTSET_FIXTURES(utTestSets)
{
	new_TestSet(Set_SetupTeardown),
};
UNTITTEST_TESTSET_HANDLER();
```

- AxisMgr.typ (reference to Logical/MachineControl/AppAxis_1/AppAxis_1/AxisMgr.typ)

### Program Logical/MachineControl/AxisTemplate/AxisMgr (IEC) - Axis control

#### AxisMgr.st - Init, cyclic, exit code
```iecst
//***********************************************************************
// Copyright: B&R Industrial Automation GmbH
// Author: B&R Industrial Automation GmbH
// Created: April 12, 2022
// Description: Tasks for axis control.
//***********************************************************************

PROGRAM _INIT

	// Read current task name for category setup
	ST_name(0, ADR(AxisControl.Status.TaskName), 0);

	// Call initialization actions
	RecipeInit;
	ConfigurationInit;
	ParameterInit;
	AxisInit;

	// Enable mapp function blocks
	MpAlarmXCore_0.Enable := TRUE;
	MpAxisBasic_0.Enable := TRUE;

END_PROGRAM

PROGRAM _CYCLIC

    MpAxisBasic_0.MpLink := ADR(gAxisTemplate);
    MC_BR_CheckRestorePositionData_0.Axis := ADR(gAxisTemplate);

	// Call all actions
    SimulationControl;
    AxisStateMachine;
    AxisCyclic;
	RecipeCyclic;

    // Assign MpLink
    MpAlarmXCore_0.MpLink := ADR(gAlarmXCore_AxisTemplate);

	// Call function block
	MpAlarmXCore_0();

END_PROGRAM

PROGRAM _EXIT

	// Disable the function blocls to unlink the MpLinks.
	// Do NOT disable MpAxisBasic, as this can cause problems during project transfer.
    MpRecipeRegPar_Par.Enable := FALSE;
	MpRecipeRegPar_Cfg.Enable := FALSE;
	MpAlarmXCore_0.Enable := FALSE;

	// Call function blocks
	MpRecipeRegPar_Par();
	MpRecipeRegPar_Cfg();
	MpAlarmXCore_0();

END_PROGRAM
```

#### AxisControlModes.st - Code that is specific to this axis
```iecst
ACTION AxisInit:
    // Action call during init
END_ACTION

ACTION AxisCyclic:
	// Cyclic action call
    IF (MpRecipeRegPar_Par.UpdateNotification) THEN

    END_IF

END_ACTION

ACTION AxisManual:
    // Action handling manual axis control
    MpAxisParameters.Jog.Velocity := AxisControl.Parameters.JogVelocity;
    MpAxisParameters.Position := AxisControl.Parameters.Position;
    MpAxisParameters.Distance := AxisControl.Parameters.Distance;
    MpAxisParameters.Acceleration := AxisControl.Parameters.Acceleration;
    MpAxisParameters.Deceleration := AxisControl.Parameters.Deceleration;

    CASE ManualState OF
		// Wait state
        MANUAL_STATE_IDLE:
            IF ((AxisControl.Command.JogNegative = TRUE) OR (AxisControl.Command.JogPositive = TRUE)) THEN
                ManualState := MANUAL_STATE_JOG;
            ELSIF ((AxisControl.Command.MoveAbsolute = TRUE) OR (AxisControl.Command.MoveAdditive = TRUE)) THEN
                MpAxisBasic_0.MoveAbsolute := AxisControl.Command.MoveAbsolute;
                MpAxisBasic_0.MoveAdditive := AxisControl.Command.MoveAdditive;
                AxisControl.Command.MoveAbsolute := FALSE;
                AxisControl.Command.MoveAdditive := FALSE;
                ManualState := MANUAL_STATE_MOVE;
            END_IF
        // Jog state
        MANUAL_STATE_JOG:
            MpAxisBasic_0.JogNegative := AxisControl.Command.JogNegative;
            MpAxisBasic_0.JogPositive := AxisControl.Command.JogPositive;
            IF (AxisControl.Command.Stop = TRUE) THEN
                AxisControl.Command.Stop := FALSE;
                MpAxisBasic_0.Stop := TRUE;
                ManualState := MANUAL_STATE_STOPPING;
            ELSIF ((AxisControl.Command.JogNegative = FALSE) AND (AxisControl.Command.JogPositive = FALSE)) THEN
                MpAxisBasic_0.Stop := FALSE;
                MpAxisBasic_0.JogPositive := FALSE;
                MpAxisBasic_0.JogNegative := FALSE;
                ManualState := MANUAL_STATE_STOPPING;
            END_IF
        // Direct move state
        MANUAL_STATE_MOVE:
            IF (AxisControl.Command.Stop = TRUE) THEN
                MpAxisBasic_0.MoveAbsolute := FALSE;
                MpAxisBasic_0.MoveAdditive := FALSE;
                AxisControl.Command.Stop := FALSE;
                MpAxisBasic_0.Stop := TRUE;
                ManualState := MANUAL_STATE_STOPPING;
            ELSIF (InPositionEdgePos.Q = TRUE) THEN
                MpAxisBasic_0.MoveAbsolute := FALSE;
                MpAxisBasic_0.MoveAdditive := FALSE;
                ManualState := MANUAL_STATE_IDLE;
                state := STATE_READY;
            ELSIF ((AxisControl.Command.JogNegative = TRUE) OR (AxisControl.Command.JogPositive = TRUE)) THEN
                MpAxisBasic_0.MoveAbsolute := FALSE;
                MpAxisBasic_0.MoveAdditive := FALSE;
                ManualState := MANUAL_STATE_JOG;
            END_IF
        // Stopping active movements
        MANUAL_STATE_STOPPING:
            MpAxisBasic_0.JogNegative := FALSE;
            MpAxisBasic_0.JogPositive := FALSE;
            MpAxisBasic_0.MoveAbsolute := FALSE;
            MpAxisBasic_0.MoveAdditive := FALSE;

            IF (MpAxisBasic_0.MoveActive = FALSE) THEN
                ManualState := MANUAL_STATE_IDLE;
                state := STATE_READY;
            END_IF
    END_CASE

END_ACTION

ACTION AxisAutomatic:
	// Action handling automatic mode
    CASE AutomaticState OF
		// Wait state
        AUTOMATIC_STATE_IDLE:
            IF (AxisControl.Command.Start = TRUE) THEN
                MpAlarmXControl_SpeedNotSet.Set := (MpAxisParameters.Velocity = 0);
                AxisControl.Command.Start := FALSE;
                AutomaticState := AUTOMATIC_STATE_RUNNING;
            END_IF
        // Automatic mode commands
        AUTOMATIC_STATE_RUNNING:
            MpAxisBasic_0.MoveVelocity := TRUE;
            MpAxisParameters.Velocity := AxisControl.Parameters.Velocity;
            MpAxisParameters.Acceleration := AxisControl.Parameters.Acceleration;
            MpAxisParameters.Deceleration := AxisControl.Parameters.Deceleration;

            IF (AxisControl.Command.Stop = TRUE) THEN
                AxisControl.Command.Stop := FALSE;
                MpAxisBasic_0.MoveVelocity := FALSE;
                state := STATE_READY;
                AutomaticState := AUTOMATIC_STATE_IDLE;
            END_IF
    END_CASE

END_ACTION

ACTION AxisReset:

END_ACTION
```

### Package Logical/MachineControl/AxisTemplate/UnitTests - Multiple variants of valid test sets

### Program Logical/MachineControl/AxisTemplate/UnitTests/prototypeTest (ANSIC) - Prototype for unit tests

#### Set_SetupTeardown.c
```c
/********************************************************************
 * COPYRIGHT --
 ********************************************************************
 * Program: -
 * Author:
 * Created:
 ********************************************************************
 * Tests for ...
 ********************************************************************/

#include <bur/plctypes.h>

#ifdef _DEFAULT_INCLUDES
#include <AsDefault.h>
#endif

#include <stdbool.h>
#include "UnitTest.h"

_SETUP_SET(void)
{
    // wait until the axis is ready
    TEST_BUSY_CONDITION(AxisControl.Status.IsReady == false);

    TEST_DONE;
}

_TEARDOWN_SET(void)
{
	TEST_DONE;
}

_SETUP_TEST(void)
{
    testState = TEST_STATE_ARRANGE;
	TEST_DONE;
}

_TEARDOWN_TEST(void)
{
    AxisControl.Command.JogNegative = false;
    AxisControl.Command.JogPositive = false;
    AxisControl.Command.MoveToStart = false;
    AxisControl.Command.Start = false;
    TEST_BUSY_CONDITION(AxisControl.Status.Velocity > 0.001);
    TEST_BUSY_CONDITION(AxisControl.Status.Velocity < -0.001);

	TEST_DONE;
}

_TEST powerOnTest(void)
{
    TEST_ABORT_CONDITION(AxisControl.Status.ErrorActive);

    switch (testState)
    {
        case TEST_STATE_ARRANGE:
            // Arrange
            AxisControl.Command.Power = true;
            TEST_BUSY_CONDITION(AxisControl.Status.Busy == false);
            testState = TEST_STATE_ACT;
            break;

        case TEST_STATE_ACT:
            // Act
            TEST_BUSY_CONDITION(AxisControl.Status.Busy);
            testState = TEST_STATE_ASSERT;
            break;

        case TEST_STATE_ASSERT:
            // Assert
            TEST_ASSERT(AxisControl.Status.IsPowered);
            testState = TEST_STATE_DONE;
            break;

        case TEST_STATE_DONE:
            /* test is done */
            TEST_DONE;
    }

    TEST_BUSY;
}

_TEST homeTest(void)
{
    TEST_ABORT_CONDITION(AxisControl.Status.ErrorActive);

    switch (testState)
    {
        case TEST_STATE_ARRANGE:
            // Arrange
            AxisControl.Command.Reference = true;
            TEST_BUSY_CONDITION(AxisControl.Status.Busy == false);
            testState = TEST_STATE_ACT;
            break;

        case TEST_STATE_ACT:
            // Act
            TEST_BUSY_CONDITION(AxisControl.Status.Busy);
            testState = TEST_STATE_ASSERT;
            break;

        case TEST_STATE_ASSERT:
            // Assert
            TEST_ASSERT(AxisControl.Status.IsHomed);
            testState = TEST_STATE_DONE;
            break;

        case TEST_STATE_DONE:
            /* test is done */
            TEST_DONE;
    }

    TEST_BUSY;
}

_TEST jogNegativeTest(void)
{
    TEST_ABORT_CONDITION(AxisControl.Status.ErrorActive);

    switch (testState)
    {
        case TEST_STATE_ARRANGE:
            // Arrange
            AxisControl.Parameters.JogVelocity = 5.0;
            testState = TEST_STATE_ACT;
            break;

        case TEST_STATE_ACT:
            // Act
            AxisControl.Command.JogNegative = true;
            TEST_BUSY_CONDITION(AxisControl.Status.Velocity > -0.01);
            testState = TEST_STATE_ASSERT;
            break;

        case TEST_STATE_ASSERT:
            // Assert
            TEST_ASSERT_REAL_WITHIN(0.01, -5.0, AxisControl.Status.Velocity);
            AxisControl.Command.JogNegative = false;
            testState = TEST_STATE_DONE;
            break;

        case TEST_STATE_DONE:
            /* test is done */
            TEST_DONE;
    }

    TEST_BUSY;
}

_TEST jogPositiveTest(void)
{
    TEST_ABORT_CONDITION(AxisControl.Status.ErrorActive);

    switch (testState)
    {
        case TEST_STATE_ARRANGE:
            // Arrange
            AxisControl.Parameters.JogVelocity = 6.0;
            testState = TEST_STATE_ACT;
            break;

        case TEST_STATE_ACT:
            // Act
            AxisControl.Command.JogPositive = true;
            TEST_BUSY_CONDITION(AxisControl.Status.Velocity < 0.01);
            testState = TEST_STATE_ASSERT;
            break;

        case TEST_STATE_ASSERT:
            // Assert
            TEST_ASSERT_REAL_WITHIN(0.01, 6.0, AxisControl.Status.Velocity);
            AxisControl.Command.JogPositive = false;
            testState = TEST_STATE_DONE;
            break;

        case TEST_STATE_DONE:
            /* test is done */
            TEST_DONE;
    }

    TEST_BUSY;
}

/*
B+R UnitTest: This is generated code.
Do not edit! Do not move!
Description: UnitTest Testprogramm infrastructure (TestSet).
LastUpdated: 2021-09-29 12:12:33Z
By B+R UnitTest Helper Version: 2.0.1.59
*/
UNITTEST_FIXTURES(fixtures)
{
	new_TestFixture("powerOnTest", powerOnTest),
	new_TestFixture("homeTest", homeTest),
	new_TestFixture("jogNegativeTest", jogNegativeTest),
	new_TestFixture("jogPositiveTest", jogPositiveTest),
};

UNITTEST_CALLER_COMPLETE_EXPLICIT(Set_SetupTeardown, "Set_SetupTeardown", setupTest, teardownTest, fixtures, setupSet, teardownSet, 0);
```

### Program Logical/MachineControl/CrossCutter/CrossCutter (IEC)

#### AxisControl.typ - Local data types
```iecst
TYPE
	AxisMachineSettingsType : {REDUND_UNREPLICABLE} 	STRUCT
		ReferencePosition : {REDUND_UNREPLICABLE} LREAL := 0.0; (*[deg] Position when the axis is referenced*)
		AxisFeatures : {REDUND_UNREPLICABLE} ARRAY[0..2]OF STRING[255] := ['CamAut_cutting',''];
		DriveConfiguration : {REDUND_UNREPLICABLE} McCfgPureVAxType := (0);
		BaseConfiguration : {REDUND_UNREPLICABLE} McCfgAxType;
	END_STRUCT;
	AxisControlCommandType : {REDUND_UNREPLICABLE} 	STRUCT
		UpdatePreviewParameters : {REDUND_UNREPLICABLE} BOOL;
		ResetEditParameters : {REDUND_UNREPLICABLE} BOOL;
		Power : {REDUND_UNREPLICABLE} BOOL;
		Reference : {REDUND_UNREPLICABLE} BOOL;
		MoveToStart : {REDUND_UNREPLICABLE} BOOL;
		MoveAbsolute : {REDUND_UNREPLICABLE} BOOL;
		MoveAdditive : {REDUND_UNREPLICABLE} BOOL;
		Abort : {REDUND_UNREPLICABLE} BOOL;
		Stop : {REDUND_UNREPLICABLE} BOOL;
		Reset : {REDUND_UNREPLICABLE} BOOL;
		JogPositive : {REDUND_UNREPLICABLE} BOOL;
		JogNegative : {REDUND_UNREPLICABLE} BOOL;
		Start : {REDUND_UNREPLICABLE} BOOL;
	END_STRUCT;
	AxisControlParametersType : {REDUND_UNREPLICABLE} 	STRUCT
		HomePosition : {REDUND_UNREPLICABLE} LREAL := 0;
		Position : {REDUND_UNREPLICABLE} LREAL := 0;
		Distance : {REDUND_UNREPLICABLE} LREAL := 180;
		Velocity : {REDUND_UNREPLICABLE} REAL := 360;
		Acceleration : {REDUND_UNREPLICABLE} REAL := 360;
		Deceleration : {REDUND_UNREPLICABLE} REAL := 360;
		JogVelocity : {REDUND_UNREPLICABLE} REAL := 360;
		StopDeceleration : {REDUND_UNREPLICABLE} REAL := 720; (*[mm/s2] Deceleration for stopping*)
		SyncAngle : {REDUND_UNREPLICABLE} LREAL := 45; (*Product Number*)
		DistanceFromSensorToCut : {REDUND_UNREPLICABLE} LREAL := 100; (*Real Product Length*)
		NumberOfKnives : {REDUND_UNREPLICABLE} USINT := 2;
		ProductLength : {REDUND_UNREPLICABLE} LREAL := 70;
		MinPrintMarkLength : {REDUND_UNREPLICABLE} LREAL := 7; (*[mm] Minimum product length, used for product detection*)
		MaxPrintMarkLength : {REDUND_UNREPLICABLE} LREAL := 15; (*[mm] Minimum print mark length, used for product detection*)
	END_STRUCT;
	AxisControlStatusType : {REDUND_UNREPLICABLE} 	STRUCT
		TaskName : {REDUND_UNREPLICABLE} STRING[80];
		MachineSettingsName : {REDUND_UNREPLICABLE} STRING[255];
		ProductSettingsName : {REDUND_UNREPLICABLE} STRING[255];
		ProductPreviewSettingsName : {REDUND_UNREPLICABLE} STRING[255];
		Status : {REDUND_UNREPLICABLE} STRING[80]; (*Machine Status*)
		IsReady : {REDUND_UNREPLICABLE} BOOL;
		ErrorActive : {REDUND_UNREPLICABLE} BOOL;
		Busy : {REDUND_UNREPLICABLE} BOOL;
		ReferenceRequired : {REDUND_UNREPLICABLE} BOOL;
		Position : {REDUND_UNREPLICABLE} LREAL;
		Velocity : {REDUND_UNREPLICABLE} REAL;
		Current : {REDUND_UNREPLICABLE} REAL;
		LagError : {REDUND_UNREPLICABLE} LREAL;
		MotorTemperature : {REDUND_UNREPLICABLE} REAL;
		IsHomed : {REDUND_UNREPLICABLE} BOOL;
		IsPowered : {REDUND_UNREPLICABLE} BOOL;
		ActualProductLength : {REDUND_UNREPLICABLE} LREAL;
		ValidProducts : {REDUND_UNREPLICABLE} UDINT;
	END_STRUCT;
	AxisControlType : {REDUND_UNREPLICABLE} 	STRUCT
		Command : {REDUND_UNREPLICABLE} AxisControlCommandType;
		Parameters : {REDUND_UNREPLICABLE} AxisControlParametersType;
		Status : {REDUND_UNREPLICABLE} AxisControlStatusType;
	END_STRUCT;
	stateEnum :
		(
		STATE_INIT,
		STATE_POWER_ON,
		STATE_HOME,
		STATE_REFERENCE,
		STATE_MOVE_TO_HOME_POSITION,
		STATE_READY,
		STATE_MANUAL_OPERATION,
		STATE_AUTOMATIC_OPERATION,
		STATE_STOPPING,
		STATE_STOPPED,
		STATE_ABORTING,
		STATE_ABORTED,
		STATE_CLEARING,
		STATE_RESETTING
		);
	configurationStateEnum :
		(
		CONFIG_STATE_INIT,
		CONFIG_STATE_READ,
		CONFIG_STATE_WRITE,
		CONFIG_STATE_READY
		);
	manualStateEnum :
		(
		MANUAL_STATE_IDLE,
		MANUAL_STATE_JOG,
		MANUAL_STATE_MOVE,
		MANUAL_STATE_STOPPING
		);
	RegistrationStatusType : {REDUND_UNREPLICABLE} 	STRUCT
		ActualMarkPosition : {REDUND_UNREPLICABLE} LREAL;
		MarkPositionError : {REDUND_UNREPLICABLE} LREAL;
		ActualProductLength : {REDUND_UNREPLICABLE} LREAL;
		ActualIntervalLength : {REDUND_UNREPLICABLE} LREAL;
		PhaseShift : {REDUND_UNREPLICABLE} LREAL;
		LastValidMarks : {REDUND_UNREPLICABLE} UDINT;
		Configuration : {REDUND_UNREPLICABLE} MpRegMarkDetectionConfigType;
	END_STRUCT;
END_TYPE
```

#### Variables.var - Local variables
```iecst
VAR
	McCamAutPar : {REDUND_UNREPLICABLE} McAcpAxCamAutParType; (*Cam automat parameters*)
	MC_BR_CamAutomatGetParFB : {REDUND_UNREPLICABLE} MC_BR_CamAutomatGetPar_AcpAx; (*Get Cam Automat Parameters Function Block*)
	MC_BR_CamAutomatSetParFB : {REDUND_UNREPLICABLE} MC_BR_CamAutomatSetPar_AcpAx; (*Set Cam Automat Parameters Function Block*)
	MC_BR_CamAutomatCommandFB : {REDUND_UNREPLICABLE} MC_BR_CamAutomatCommand;
	MpRegMarkDetectionFB : {REDUND_UNREPLICABLE} MpRegMarkDetection;
	MpRegMarkDetectionConfigFB : {REDUND_UNREPLICABLE} MpRegMarkDetectionConfig;
	RegistrationControl : {REDUND_UNREPLICABLE} RegistrationStatusType;
	MC_BR_PhasingFB : {REDUND_UNREPLICABLE} MC_BR_Phasing;
	MpAlarmXControlProductLengthFB : {REDUND_UNREPLICABLE} MpAlarmXAlarmControl;
END_VAR
```

#### ManualCommand.st
```iecst
// Returns True if a manual command is active, false otherwise
FUNCTION ManualCommand
    ManualCommand := Commands.JogNegative OR Commands.JogPositive OR Commands.MoveAbsolute OR Commands.MoveAdditive;
END_FUNCTION
```

### Package Logical/MachineControl/CrossCutter/UnitTests - Multiple variants of valid test sets

### Program Logical/MachineControl/CrossCutter/UnitTests/CutterTest (ANSIC) - Prototype for unit tests

#### variables.var
```iecst
(********************************************************************
 * COPYRIGHT --
 ********************************************************************
 * Program: utTemplate_automated
 * File: variables.var
 * Author: -
 * Created: -
 ********************************************************************
 * Local variables of program utTemplate_automated
 ********************************************************************)
(*Describe the test*)
VAR
	Testsuite : {REDUND_UNREPLICABLE} UtMgrTestSuite := (Name:='prototype',Description:='automated tests for cross cutter axis',Type:=utMgrTEST_TYPE_C);
	lastTestCase : {REDUND_UNREPLICABLE} STRING[80];
	lastTestSet : {REDUND_UNREPLICABLE} STRING[80];
END_VAR
(*Variables used in the tests*)
VAR
	AxisControl : {REDUND_UNREPLICABLE} AxisControlType;
	absVelocity : {REDUND_UNREPLICABLE} REAL;
	testState : {REDUND_UNREPLICABLE} testState_enum;
END_VAR
```

#### testSuite.c
```c
/********************************************************************
 * COPYRIGHT --
 ********************************************************************
 * Program: -
 * Author:
 * Created:
 ********************************************************************
 * Test registration and handshake
 ********************************************************************/

#include <bur/plctypes.h>

#ifdef _DEFAULT_INCLUDES
#include <AsDefault.h>
#endif

#include "UnitTest.h"
#include <string.h>

void _INIT initTestSuite(void)
{
	utInit(&Testsuite);
}

void _CYCLIC cyclicWithTest(void)
{
	utCyclic(&Testsuite);

    if (Testsuite.Informational.LastKnownPassedLocation.TestCaseName != 0)
        strcpy((char*)&lastTestCase, (char*)Testsuite.Informational.LastKnownPassedLocation.TestCaseName);
    if (Testsuite.Informational.LastKnownPassedLocation.TestSetName != 0)
        strcpy((char*)&lastTestSet, (char*)Testsuite.Informational.LastKnownPassedLocation.TestSetName);
}

void _EXIT exitTestSuite(void)
{
	utExit(&Testsuite);
}
```

### Program Logical/MainControl/MainCtrl (IEC)

#### Main.st - Init, cyclic, exit code
```iecst
//*********************************************************************************
//* Copyright: B&R Industrial Automation GmbH
//* Author:    B&R Industrial Automation GmbH
//* Created:   30. Sep 2020/08:00
//* Description: Tasks for axis control. The Main Cross Cutter handling is done in this task.
//*********************************************************************************

PROGRAM _INIT
	// Register parameters to MpRecipe
	MpRecipeRegPar_M.MpLink := ADR(gMpLinkRecipeXml);
	MpRecipeRegPar_M.Enable := TRUE;
	MpRecipeRegPar_M.Category := ADR('Machine Configuration');
	MpRecipeRegPar_M.PVName := ADR('MainCtrl:MainCtrl.FixPar');
	MpRecipeRegPar_P.MpLink := ADR(gMpLinkRecipeXml);
	MpRecipeRegPar_P.Enable := TRUE;
	MpRecipeRegPar_P.Category := ADR('Parameters');
	MpRecipeRegPar_P.PVName := ADR('MainCtrl:MainCtrl.Para');
	MpRecipeRegPar_Pre1.MpLink := ADR(gRecipeXmlPreviewMpLink);
	MpRecipeRegPar_Pre1.Enable := TRUE;
	MpRecipeRegPar_Pre1.Category := ADR('Preview');
	MpRecipeRegPar_Pre1.PVName := ADR('MainCtrl:PreviewParameters');
	MpRecipeRegPar_Pre2.MpLink := ADR(gMpLinkRecipeXml);
	MpRecipeRegPar_Pre2.Enable := TRUE;
	MpRecipeRegPar_Pre2.Category := ADR('Parameters');
	MpRecipeRegPar_Pre2.PVName := ADR('MainCtrl:PreviewParameters');

	// Activate RegPar FUBs
	WHILE NOT MpRecipeRegPar_M.Active DO
		MpRecipeRegPar_M();
	END_WHILE
	WHILE NOT MpRecipeRegPar_P.Active DO
		MpRecipeRegPar_P();
	END_WHILE
	WHILE NOT MpRecipeRegPar_Pre1.Active DO
		MpRecipeRegPar_Pre1();
	END_WHILE
    WHILE NOT MpRecipeRegPar_Pre2.Active DO
		MpRecipeRegPar_Pre2();
	END_WHILE

    // Init Cam automat related function blocks ***************************************
	InitCamAutFunctionBlocks;

	// Axis No.0 initialization *********************************************************************************
	MpAxisBasic_x[0].MpLink := ADR(gAxisMaster);
	MpAxisBasic_x[0].Enable := TRUE;
	MpAxisBasic_x[0].Parameters := ADR(AxisControl[0].Parameter.AxPar);
	MC_ReadAxisError_x[0].Axis := ADR(gAxisMaster);
	MC_ReadActualTorque_x[0].Axis := ADR(gAxisMaster);

	// Axis No.1 initialization *********************************************************************************
	MpAxisBasic_x[1].MpLink := ADR(gAxisSlave);
	MpAxisBasic_x[1].Enable := TRUE;
	MpAxisBasic_x[1].Parameters := ADR(AxisControl[1].Parameter.AxPar);
	MC_ReadAxisError_x[1].Axis := ADR(gAxisSlave);
	MC_ReadActualTorque_x[1].Axis := ADR(gAxisSlave);
END_PROGRAM

PROGRAM _CYCLIC

	//******************** Init cam automat parameters ********************
	GetCamAutPar;

	//******************** Axis status updates ********************
	//******************** Status information is read before the state machine to attain a shorter reaction time in case of error ********************
	AxisStatusUpdate;

	//******************** Axis control ********************
	AxisStateMachine;

	//******************** Crosscutter control ********************
	CrossCutter;

	//*************************************************

	//******************** Copy preview parameters before creating or saving a recipe ********************
	IF CopyPreviewParameters THEN
		PreviewParameters := MainCtrl.Parameter;
		CopyPreviewParameters := FALSE;
	END_IF
	IF ResetEditValues THEN
		MainCtrl.Parameter := PreviewParameters;
		ResetEditValues := FALSE;
    END_IF

	//******************** MpAxisBasic function block calls ********************
	FOR AxIndex := 0 TO MAX_IDX_AXIS DO
		MpAxisBasic_x[AxIndex]();
	END_FOR

	//******************** CamAutomat function block calls ********************
	MC_BR_CamAutomatSetPar_AcpAx_0();
	MC_BR_CamAutomatGetPar_AcpAx_0();
	MC_BR_CamAutomatCommand_0();

	//******************** MpRecipeRegPar FB calls ********************
	MpRecipeRegPar_M();
	MpRecipeRegPar_P();
	MpRecipeRegPar_Pre1();
	MpRecipeRegPar_Pre2();
END_PROGRAM

PROGRAM _EXIT
	MpRecipeRegPar_M.Enable := FALSE;
	MpRecipeRegPar_M();
	MpRecipeRegPar_P.Enable := FALSE;
	MpRecipeRegPar_P();
	MpRecipeRegPar_Pre1.Enable := FALSE;
	MpRecipeRegPar_Pre1();
	MpRecipeRegPar_Pre2.Enable := FALSE;
	MpRecipeRegPar_Pre2();
	FOR AxIndex := 0 TO MAX_IDX_AXIS DO
		MpAxisBasic_x[AxIndex].Enable := FALSE;
		MpAxisBasic_x[AxIndex]();
	END_FOR
END_PROGRAM
```

#### Variables.var - Local variables
```iecst
(*Main Control*)
VAR
	MainCtrl : MainCtrlType; (*Main Control Variable*)
	MpAxisBasic_x : ARRAY[0..MAX_IDX_AXIS] OF MpAxisBasic; (*MpAxis Declaration*)
	PreviewParameters : MainParametersType;
	MpRecipeRegPar_M : MpRecipeRegPar; (*Register fix parameters to MpRecipe*)
	MpRecipeRegPar_Pre1 : MpRecipeRegPar; (*Register preview parameters*)
	MpRecipeRegPar_Pre2 : MpRecipeRegPar; (*Register preview parameters*)
	MpRecipeRegPar_P : MpRecipeRegPar; (*Register product parameters to MpRecipe*)
	ReactionName : STRING[80]; (*String to check for MpAlarmX reactions*)
	LastAutoModeOn : BOOL; (*Last cycle's status of auto mode on switch*)
	ResetEditValues : BOOL;
	CopyPreviewParameters : BOOL;
END_VAR
(*Motion Control Related Variables*)
VAR
	AxisControl : ARRAY[0..MAX_IDX_AXIS] OF AxControlType; (*control structure*)
	McCamAutDefine : McAcpAxCamAutDefineType; (*Definition of cam automat parameters*)
	McCamAutPar : McAcpAxCamAutParType; (*Cam automat parameters*)
	MC_ReadAxisError_x : ARRAY[0..MAX_IDX_AXIS] OF MC_ReadAxisError; (*Read Axis Error Function Block*)
	MC_ReadActualTorque_x : ARRAY[0..MAX_IDX_AXIS] OF MC_ReadActualTorque; (*Read Actual PositionFunction Block *)
	MC_BR_CamAutomatCommand_0 : MC_BR_CamAutomatCommand; (*Cam Automat Command Function Block*)
	MC_BR_CamAutomatGetPar_AcpAx_0 : MC_BR_CamAutomatGetPar_AcpAx; (*Get Cam Automat Parameters Function Block*)
	MC_BR_CamAutomatSetPar_AcpAx_0 : MC_BR_CamAutomatSetPar_AcpAx; (*Set Cam Automat Parameters Function Block*)
	StopMovementsReaction : BOOL; (*Stop movements on positive edge of alarm reaction*)
	AxIndex : USINT := 0; (*Index for Axis in FOR Statement*)
	InitCamAut : USINT; (*state of initializing camaut data*)
	UpdateCamAutomat : BOOL;
	CamUpdateState : USINT;
END_VAR
(*Constants*)
VAR CONSTANT
	AXIS_IDX_FEEDER : USINT := 0; (*Axis index of the feeder axis*)
	AXIS_IDX_CUTTER : USINT := 1; (*Axis index of the cutter axis*)
	MAX_IDX_AXIS : USINT := 1; (*Max axis index*)
END_VAR
```

#### CamAutomatActions.st
```iecst
//*********************************************************************************
//* Copyright: B&R Industrial Automation GmbH
//* Author:    B&R Industrial Automation GmbH
//* Created:   24 June, 2021/15:05
//* This task reads the cam automat data from the ACOPOS into the PV structure
//*********************************************************************************

ACTION InitCamAutFunctionBlocks:
	// Init cam automat related function blocks
	McCamAutDefine.DataAddress := ADR(McCamAutPar);
	MC_BR_CamAutomatGetPar_AcpAx_0.Slave := ADR(gAxisSlave);
	MC_BR_CamAutomatGetPar_AcpAx_0.Command := mcGET_PAR_ACTUAL;
	MC_BR_CamAutomatGetPar_AcpAx_0.CamAutomat := McCamAutDefine;
    MC_BR_CamAutomatSetPar_AcpAx_0.Command := mcSET_UPDATE_FROM_ADR;
    // Synchron means the new parameters are valid when an event with synchronous update = TRUE happens
	MC_BR_CamAutomatSetPar_AcpAx_0.AdvancedParameters.ParLock := mcCAMAUT_UNLOCK_SYNCHRON;
	MC_BR_CamAutomatSetPar_AcpAx_0.CamAutomat := McCamAutDefine;
	MC_BR_CamAutomatSetPar_AcpAx_0.Slave := ADR(gAxisSlave);
	MC_BR_CamAutomatCommand_0.Slave := ADR(gAxisSlave);
	MC_BR_CamAutomatCommand_0.Enable := TRUE;
END_ACTION

ACTION GetCamAutPar:
	CASE InitCamAut OF
		0: // Set up function blocks for reading and writing cam automat parameters
			MC_BR_CamAutomatGetPar_AcpAx_0.Execute := TRUE;
			InitCamAut := 1;

		1: // Wait for function block done
			IF MC_BR_CamAutomatGetPar_AcpAx_0.Done THEN
				MC_BR_CamAutomatGetPar_AcpAx_0.Execute := FALSE;
				InitCamAut := 10;
			END_IF
			// In case of error abort reading
			IF MC_BR_CamAutomatGetPar_AcpAx_0.Error THEN
				MC_BR_CamAutomatGetPar_AcpAx_0.Execute := FALSE;
				InitCamAut := 100;
			END_IF

		10: // Done, do nothing

		100: // Error handling
	END_CASE;
END_ACTION

ACTION UpdateCamAutomatAction:
	CASE CamUpdateState OF
		0: // Calculate new cam automat parameters
			IF UpdateCamAutomat AND (InitCamAut = 10) THEN
				// General CAM settings
				McCamAutPar.Common.Master.MasterStartInterval := MainCtrl.Intern.ProductLength[MainCtrl.Status.CurrentBatch];
				McCamAutPar.Common.Master.MasterStartPosition := 0;

				// CAM state 0: Base state, wait for master start position
				McCamAutPar.State[0].Event[0].NextState := 1;
				McCamAutPar.State[0].Event[0].SynchronousUpdate := mcSWITCH_ON;
                McCamAutPar.State[0].Event[0].Transition := mcEVENT_IMMEDIATELY;
                // Starts cutting process on interval, modify according to machine e.g. change to mcEVENT_SRC_TRIGGER1 for a signal wired to input channel 1 on ACOPOS
				McCamAutPar.State[0].Event[0].Type := mcEVENT_START_POSITION;

                // CAM state 1: First cut movement
                // * 100 because of measurement units to resolution units conversion
                McCamAutPar.State[1].MasterFactor := REAL_TO_DINT(GatDegreeToDistance(MainCtrl.FixParameter.SyncAngle, MainCtrl.FixParameter.CutDiameter / 2) * 100);
                // * 100 because of measurement units to resolution units conversion
                McCamAutPar.State[1].SlaveFactor := REAL_TO_DINT(MainCtrl.FixParameter.SyncAngle * 100);
                // Assuming print mark signals coincide with cutting positions
				McCamAutPar.State[1].CompensationParameters.MasterCompDistance := MainCtrl.Intern.ProductLength[MainCtrl.Status.CurrentBatch];
				IF MainCtrl.FixParameter.NrOfKnives = 0 THEN
					// There must be at least one knife!
					MainCtrl.FixParameter.NrOfKnives := 1;
				END_IF
				McCamAutPar.State[1].CompensationParameters.SlaveCompDistance := (360 / (2 * MainCtrl.FixParameter.NrOfKnives)) - (MainCtrl.FixParameter.SyncAngle / 2);
				// Change to next state at end of state
				McCamAutPar.State[1].Event[0].NextState := 3;
				McCamAutPar.State[1].Event[0].SynchronousUpdate := mcSWITCH_ON;
				McCamAutPar.State[1].Event[0].Transition := mcEVENT_END_OF_STATE;
				McCamAutPar.State[1].Event[0].Type := mcEVENT_SIGNAL2;
				McCamAutPar.State[1].Event[1].NextState := 2;
				McCamAutPar.State[1].Event[1].SynchronousUpdate := mcSWITCH_ON;
				McCamAutPar.State[1].Event[1].Transition := mcEVENT_END_OF_STATE;
				McCamAutPar.State[1].Event[1].Type := mcEVENT_STATE_END;

                // CAM state 2: Repeating cut movements
                // * 100 because of measurement units to resolution units conversion
				McCamAutPar.State[2].MasterFactor := REAL_TO_DINT(GatDegreeToDistance(MainCtrl.FixParameter.SyncAngle, MainCtrl.FixParameter.CutDiameter / 2) * 100);
				McCamAutPar.State[2].SlaveFactor := REAL_TO_DINT(MainCtrl.FixParameter.SyncAngle * 100);// * 100 because of measurement units to resolution units conversion
				McCamAutPar.State[2].CompensationParameters.MasterCompDistance := MainCtrl.Intern.ProductLength[MainCtrl.Status.CurrentBatch];
				McCamAutPar.State[2].CompensationParameters.SlaveCompDistance := (360 / MainCtrl.FixParameter.NrOfKnives);
				// Repeat state at end of state, or go to next state in case of signal 2 (stop cutting signal)
				McCamAutPar.State[2].Event[0].NextState := 3;
				McCamAutPar.State[2].Event[0].SynchronousUpdate := mcSWITCH_ON;
				McCamAutPar.State[2].Event[0].Transition := mcEVENT_END_OF_STATE;
				McCamAutPar.State[2].Event[0].Type := mcEVENT_SIGNAL2;
				McCamAutPar.State[2].Event[1].NextState := 2;
				McCamAutPar.State[2].Event[1].SynchronousUpdate := mcSWITCH_ON;
				McCamAutPar.State[2].Event[1].Transition := mcEVENT_END_OF_STATE;
				McCamAutPar.State[2].Event[1].Type := mcEVENT_STATE_END;

                // CAM state 3: Decelerate and stop at home position
                // Master with any positive value & slave = 0 means slave is not moving
                McCamAutPar.State[3].MasterFactor := 100;
                // Master with any positive value & slave = 0 means slave is not moving
                McCamAutPar.State[3].SlaveFactor := 0;
                // allow half a product length to stop
				McCamAutPar.State[3].CompensationParameters.MasterCompDistance := MainCtrl.Intern.ProductLength[MainCtrl.Status.CurrentBatch] / 2;
				McCamAutPar.State[3].CompensationParameters.SlaveCompDistance := (360 / (2 * MainCtrl.FixParameter.NrOfKnives));
				// Return to base state after axis has stopped
				McCamAutPar.State[3].Event[0].NextState := 0;
				McCamAutPar.State[3].Event[0].SynchronousUpdate := mcSWITCH_ON;
				McCamAutPar.State[3].Event[0].Transition := mcEVENT_END_OF_STATE;
				McCamAutPar.State[3].Event[0].Type := mcEVENT_STATE_END;

				MC_BR_CamAutomatSetPar_AcpAx_0.Execute := TRUE;
				CamUpdateState := 1;
			END_IF

		1: // Wait for SetPar done
			IF MC_BR_CamAutomatSetPar_AcpAx_0.Done THEN
				UpdateCamAutomat := FALSE;
				MC_BR_CamAutomatSetPar_AcpAx_0.Execute := FALSE;
				CamUpdateState := 0;
			ELSIF MC_BR_CamAutomatSetPar_AcpAx_0.Error THEN
				// Error handling
				MpAlarmXSet(gMpLinkAlarmXCore, 'SetCamFailed');
				UpdateCamAutomat := FALSE;
				MC_BR_CamAutomatSetPar_AcpAx_0.Execute := FALSE;
				CamUpdateState := 0;
			END_IF
	END_CASE;
END_ACTION
```

#### AxisStatusUpdate.st
```iecst
//*********************************************************************************
//* Copyright: B&R Industrial Automation GmbH
//* Created:   29 June, 2021/09:58
//* This file contains the logic to update the axis status information
//*********************************************************************************

ACTION AxisStatusUpdate:
	FOR AxIndex := 0 TO MAX_IDX_AXIS DO
		//*********************** MpAxisBasic_x information ************************
		AxisControl[AxIndex].Status.ActualPLCOpenState := MpAxisBasic_x[AxIndex].Info.PLCopenState;
		AxisControl[AxIndex].Status.MovementActive := MpAxisBasic_x[AxIndex].MoveActive;
		AxisControl[AxIndex].Status.TorqueLimited := MpAxisBasic_x[AxIndex].Info.LimitLoadActive;
		AxisControl[AxIndex].Status.ActPosition := MpAxisBasic_x[AxIndex].Position;
		AxisControl[AxIndex].Status.ActVelocity := MpAxisBasic_x[AxIndex].Velocity;
		AxisControl[AxIndex].Status.Error := MpAxisBasic_x[AxIndex].Error;
		AxisControl[AxIndex].Status.PowerOn := MpAxisBasic_x[AxIndex].PowerOn;
		AxisControl[AxIndex].Status.IsHomed := MpAxisBasic_x[AxIndex].IsHomed;

		IF MpAxisBasic_x[AxIndex].Active AND (MpAxisBasic_x[AxIndex].Info.CommunicationState = mcCOMM_STATE_ACTIVE) THEN
			//******************* MC_READACTUALTORQUE ********************
			MC_ReadActualTorque_x[AxIndex].Enable := NOT(MC_ReadActualTorque_x[AxIndex].Error);
			MC_ReadActualTorque_x[AxIndex]();
			IF MC_ReadActualTorque_x[AxIndex].Valid THEN
				AxisControl[AxIndex].Status.ActTorque := MC_ReadActualTorque_x[AxIndex].Torque;
			END_IF

			//*********************** MC_READAXISERROR *********************
			MC_ReadAxisError_x[AxIndex].Enable := NOT(MC_ReadAxisError_x[AxIndex].Error);
			MC_ReadAxisError_x[AxIndex]();
			IF MC_ReadAxisError_x[AxIndex].Valid THEN
				AxisControl[AxIndex].Status.ErrorID := MC_ReadAxisError_x[AxIndex].AxisErrorID;
			END_IF
		END_IF

		//*************** CHECK FOR GENERAL AXIS ERROR *****************
		IF ((MC_ReadAxisError_x[AxIndex].AxisErrorID <> 0) AND MC_ReadAxisError_x[AxIndex].Valid) OR MpAxisBasic_x[AxIndex].Error THEN
			// Set error state if not already in error state / or error reset state
			IF AxisControl[AxIndex].AxisState < AX_STATE_ERROR THEN
				AxisControl[AxIndex].AxisState := AX_STATE_ERROR;
			END_IF
		ELSIF AxisControl[AxIndex].AxisState < AX_STATE_ERROR THEN
			AxisControl[AxIndex].Command.ErrorAcknowledge := FALSE ;
		END_IF
	END_FOR // FOR uAxIndex := 0 TO MAX_IDX_AXIS DO
END_ACTION
```

### Program Logical/MainControl/PIDControl (IEC) - PID control task

#### Main.st - Init, cyclic, exit code
```iecst
//*********************************************************************************
//* Copyright: B&R Industrial Automation GmbH
//* Created:   22 July, 2021/15:54
//* This task contains the logic for a PID controller
//*********************************************************************************

PROGRAM _INIT
	// Register parameters to the recipe
	MpRecipeRegPar_P.MpLink := ADR(gMpLinkRecipeXml);
	MpRecipeRegPar_P.Enable := TRUE;
	MpRecipeRegPar_P.PVName := ADR('PIDControl:PidControlParameters');
	MpRecipeRegPar_P.Category := ADR('Parameters');
	MpRecipeRegPar_Pre.MpLink := ADR(gRecipeXmlPreviewMpLink);
	MpRecipeRegPar_Pre.Enable := TRUE;
	MpRecipeRegPar_Pre.PVName := ADR('PIDControl:PidControlParameters');
	MpRecipeRegPar_Pre.Category := ADR('Preview');
	// Activate recipe registration
	WHILE NOT MpRecipeRegPar_P.Active DO
		MpRecipeRegPar_P();
	END_WHILE
	WHILE NOT MpRecipeRegPar_Pre.Active DO
		MpRecipeRegPar_Pre();
	END_WHILE
	// Keep start signal of tuning fub true, tuning is started and stopped via HMI by setting the enable input
	MTBasicsOscillationTuning_0.Start := TRUE;
END_PROGRAM

PROGRAM _CYCLIC
	// Simulation
	SimulateActValue;

	// Update parameters on update notification
	IF MpRecipeRegPar_P.UpdateNotification THEN
		MTBasicsPID_0.PIDParameters := PidControlParameters.PidParameters;
		MTBasicsPID_0.SetValue := PidControlParameters.SetValue;
		MTBasicsPID_0.MinOut := PidControlParameters.MinOut;
		MTBasicsPID_0.MaxOut := PidControlParameters.MaxOut;
		MTBasicsPID_0.Invert := PidControlParameters.Invert;
		MTBasicsPID_0.Update := MTBasicsPID_0.Active;
		MTBasicsOscillationTuning_0.MinOut := PidControlParameters.MinOut;
		MTBasicsOscillationTuning_0.MaxOut := PidControlParameters.MaxOut;
		MTBasicsOscillationTuning_0.SetValue := PidControlParameters.SetValue;
		MTBasicsOscillationTuning_0.Invert := PidControlParameters.Invert;
		MTBasicsOscillationTuning_0.Update := MTBasicsOscillationTuning_0.Active;
	END_IF

	// Update actual value
	MTBasicsPID_0.ActValue := ActValue;
	MTBasicsOscillationTuning_0.ActValue := ActValue;

	// Autotuning of parameters
	IF MTBasicsOscillationTuning_0.TuningDone THEN
		PidControlParameters.PidParameters := MTBasicsOscillationTuning_0.PIDParameters;
		TuningQuality := MTBasicsOscillationTuning_0.Quality;
	END_IF

	// Reset update commands
	IF MTBasicsPID_0.UpdateDone THEN
		MTBasicsPID_0.Update := FALSE;
	ELSIF MTBasicsOscillationTuning_0.UpdateDone THEN
		MTBasicsOscillationTuning_0.Update := FALSE;
	END_IF

	// Call function blocks
	MpRecipeRegPar_P();
	MpRecipeRegPar_Pre();
	MTBasicsPID_0();
	MTBasicsOscillationTuning_0();

	// Update status value
	IF MTBasicsOscillationTuning_0.TuningActive THEN
		PidStatus := PID_TUNING;
	ELSIF MTBasicsPID_0.Error THEN
		PidStatus := PID_ERROR;
	ELSIF MTBasicsPID_0.Active THEN
		PidStatus := PID_ACTIVE;
	ELSE
		PidStatus := PID_IDLE;
	END_IF

	// Set output value
	IF MTBasicsOscillationTuning_0.TuningActive THEN
		OutValue := MTBasicsOscillationTuning_0.Out;
	ELSE
		OutValue := MTBasicsPID_0.Out;
	END_IF
END_PROGRAM

PROGRAM _EXIT
	MpRecipeRegPar_P.Enable := FALSE;
	MpRecipeRegPar_P();
	MpRecipeRegPar_Pre.Enable := FALSE;
	MpRecipeRegPar_Pre();
END_PROGRAM
```

#### Types.typ - Local data types
```iecst
TYPE
	PidStateEnum :
		(
		PID_IDLE := 0,
		PID_ACTIVE := 1,
		PID_TUNING := 2,
		PID_ERROR := 3
		);
	PidControlParametersType : 	STRUCT
		PidParameters : MTPIDParametersType;
		SetValue : REAL;
		MinOut : REAL;
		MaxOut : REAL;
		Invert : BOOL;
	END_STRUCT;
END_TYPE
```

- Machine.mcfg (not shown)

Listed in the project but not available here: Logical/Infrastructure/Audit/AuditMgr/AuditMgr.st, Logical/Infrastructure/Audit/AuditMgr/AuditMgr.typ, Logical/Infrastructure/Audit/AuditMgr/AuditMgr.var, Logical/Infrastructure/File/FileMgr/FileMgr.st, Logical/Infrastructure/File/FileMgr/FileMgr.var, Logical/Infrastructure/SysServices/IoBrowser/Main.st, Logical/Infrastructure/SysServices/IoBrowser/Types.typ, Logical/Infrastructure/SysServices/IoBrowser/mappViewAction.st, Logical/Infrastructure/TS_UnitTest/Libraries/UnitTest/include/Asserts.hpp, Logical/Infrastructure/TS_UnitTest/Libraries/UnitTest/include/TestCaller.h, Logical/Infrastructure/TS_UnitTest/Libraries/UnitTest/include/TestCase.h, Logical/Infrastructure/TS_UnitTest/Samples/Tests_Program/SPLMyCalc/SPLMyCalc.typ, Logical/Infrastructure/TS_UnitTest/Samples/Tests_Program/SPLMyCalc/SPLMyCalc.var, Logical/Infrastructure/TS_UnitTest/Samples/Tests_Program/SPLMyCalc/SPLMyCalc.fun, Logical/Infrastructure/TS_UnitTest/Samples/Tests_Program/Tests_MyCalcLib_C/SPL_CalcTest/variables.var, Logical/Infrastructure/TS_UnitTest/Samples/Tests_Program/Tests_MyCalcLib_C/SPL_CalcTest/autoGeneratedFile.c, Logical/Infrastructure/TS_UnitTest/Samples/Tests_Program/Tests_MyCalcLib_C/SPL_CalcTest/testSet_MyCalcLib_Subtraction.c, Logical/Infrastructure/TS_UnitTest/Samples/Tests_Program/Tests_MyCalcLib_C/SPL_CalcTest_Variants/testSuite.c, Logical/Infrastructure/TS_UnitTest/Samples/Tests_Program/Tests_MyCalcLib_C/SPL_CalcTest_Variants/autoGeneratedFile.c, Logical/Infrastructure/TS_UnitTest/Samples/Tests_Program/Tests_MyCalcLib_C/SPL_CalcTest_Variants/testSet_MyCalcLib_Subtraction.c, Logical/Infrastructure/TS_UnitTest/Samples/Tests_Program/Tests_MyCalcLib_C/SPL_CalcTest_Variants/testSet_MyCalcLib_Subtraction_variantA.c, Logical/Infrastructure/TS_UnitTest/Samples/Tests_Program/Tests_MyCalcLib_C/SPL_CalcTest_Variants/testSet_MyCalcLib_Subtraction_variantB.c, Logical/Infrastructure/TS_UnitTest/Samples/Tests_Program/Tests_MyCalcLib_C/SPL_CalcTest_Variants/testSet_MyCalcLib_Subtraction_variantC.c, Logical/Infrastructure/TS_UnitTest/Samples/Tests_Program/Tests_MyCalcLib_C/SPL_CalcTest_Variants/testSet_MyCalcLib_Subtraction_variantD.c, Logical/Infrastructure/TS_UnitTest/Samples/Framework_Extension_With_Custom_Asserts/SPL_AssertsEx/testSuite.c, Logical/Infrastructure/TS_UnitTest/Samples/Framework_Extension_With_Custom_Asserts/SPL_AssertsEx/varAssertExt.var, Logical/Infrastructure/TS_UnitTest/Samples/Framework_Extension_With_Custom_Asserts/SPL_AssertsEx/testSet_AssertsExt.c, Logical/Infrastructure/TS_UnitTest/Samples/Framework_Features/SPL_Behavior/ControlFlow/test_SetTestCases.c, Logical/Infrastructure/TS_UnitTest/Samples/Framework_Features/SPL_Behavior/ControlFlow/test_SetTestCases_SetSetup_SetTeardown.c, Logical/Infrastructure/TS_UnitTest/Samples/Framework_Features/SPL_Behavior/ControlFlow/test_SetComplete.c, Logical/Infrastructure/TS_UnitTest/Templates/HelperTool_Supported/utTemplate_automated, Logical/Infrastructure/TS_UnitTest/Templates/HelperTool_Supported/TestSet_Templates/Set_Testcases.c, Logical/Infrastructure/TS_UnitTest/Templates/HelperTool_Supported/TestSet_Templates/Set_SetupTeardown.c, Logical/MachineControl/AppAxis_1/UnitTests/ConvTest/variables.var, Logical/MachineControl/AppAxis_1/UnitTests/ConvTest/testSuite.c, Logical/MachineControl/AppAxis_1/UnitTests/ConvTest/Set_SetupTeardown.c, Logical/MachineControl/AxisTemplate/AxisMgr/AxisMgr.typ, Logical/MachineControl/AxisTemplate/AxisMgr/AxisMgr.var, Logical/MachineControl/AxisTemplate/AxisMgr/Variables.var, Logical/MachineControl/AxisTemplate/AxisMgr/AxisStateMachine.st, Logical/MachineControl/AxisTemplate/AxisMgr/Recipe.st, Logical/MachineControl/AxisTemplate/AxisMgr/SimulationControl.st, Logical/MachineControl/AxisTemplate/AxisMgr/LocalFunctions.fun, Logical/MachineControl/AxisTemplate/AxisMgr/ManualCommand.st, Logical/MachineControl/AxisTemplate/AxisMgr/AutomaticCommand.st, Logical/MachineControl/AxisTemplate/AxisMgr/ChangeConfiguration.st, Logical/MachineControl/CrossCutter/CrossCutter/AxisControl.st, Logical/MachineControl/CrossCutter/CrossCutter/SimulationControl.st, Logical/MachineControl/CrossCutter/CrossCutter/AxisControlModes.st, Logical/MachineControl/CrossCutter/CrossCutter/LocalFunctions.fun, Logical/MachineControl/CrossCutter/CrossCutter/AutomaticCommand.st, Logical/MachineControl/AxisTemplate/AxisMgr/AxisMgr.var, Logical/MachineControl/AxisTemplate/AxisMgr/AxisStateMachine.st, Logical/MachineControl/AxisTemplate/AxisMgr/ChangeConfiguration.st, Logical/MachineControl/AxisTemplate/AxisMgr/Recipe.st, Logical/MainControl/MainCtrl/Types.typ, Logical/MainControl/MainCtrl/CrossCutter.st, Logical/MainControl/MainCtrl/AxisStateMachine.st, Logical/MainControl/PIDControl/Variables.var, Logical/MainControl/PIDControl/SimulateActValue.st
